LIN {X 0,Y 392.487,Z 448.569,A -85,B 0,C 180,E1 15700.156,E2 15700.156} C_VEL
LIN {X 0,Y 396.034,Z 422.526,A -85,B 0,C 180,E1 15700.091,E2 15700.091} C_VEL
LIN {X 0,Y 397.206,Z 415.686,A -85,B 0,C 180,E1 15700.071,E2 15700.071} C_VEL
LIN {X 0,Y 405.627,Z 392.982,A -85,B 0,C 180,E1 15699.396,E2 15699.396} C_VEL
LIN {X 0,Y 416.715,Z 367.074,A -85,B 0,C 180,E1 15698.867,E2 15698.867} C_VEL
LIN {X 0,Y 418.207,Z 363.431,A -85,B 0,C 180,E1 15698.784,E2 15698.784} C_VEL
LIN {X 0,Y 413.743,Z 355.491,A -85,B 0,C 180,E1 15697.429,E2 15697.429} C_VEL
LIN {X 0,Y 395.759,Z 367.716,A -85,B 0,C 180,E1 15695.526,E2 15695.526} C_VEL
LIN {X 0,Y 388.299,Z 373.214,A -85,B 0,C 180,E1 15694.685,E2 15694.685} C_VEL
LIN {X 0,Y 386.532,Z 374.791,A -85,B 0,C 180,E1 15694.506,E2 15694.506} C_VEL
LIN {X 0,Y 379.414,Z 383.98,A -85,B 0,C 180,E1 15694.055,E2 15694.055} C_VEL
LIN {X 0,Y 377.884,Z 385.781,A -85,B 0,C 180,E1 15693.937,E2 15693.937} C_VEL
LIN {X 0,Y 373.363,Z 392.757,A -85,B 0,C 180,E1 15693.757,E2 15693.757} C_VEL
LIN {X 0,Y 371.922,Z 395.3,A -85,B 0,C 180,E1 15693.628,E2 15693.628} C_VEL
LIN {X 0,Y 367.95,Z 408.603,A -85,B 0,C 180,E1 15693.013,E2 15693.013} C_VEL
LIN {X 0,Y 361.272,Z 436.616,A -85,B 0,C 180,E1 15692.192,E2 15692.192} C_VEL
LIN {X 0,Y 356.729,Z 450.848,A -85,B 0,C 180,E1 15691.567,E2 15691.567} C_VEL
LIN {X 0,Y 354.7,Z 456.048,A -85,B 0,C 180,E1 15691.213,E2 15691.213} C_VEL
LIN {X 0,Y 350.036,Z 511.042,A -85,B 0,C 180,E1 15689.32,E2 15689.32} C_VEL
LIN {X 0,Y 348.814,Z 540.503,A -85,B 0,C 180,E1 15688.156,E2 15688.156} C_VEL
LIN {X 0,Y 347.785,Z 558.819,A -85,B 0,C 180,E1 15687.108,E2 15687.108} C_VEL
LIN {X 0,Y 346.431,Z 575.545,A -85,B 0,C 180,E1 15685.836,E2 15685.836} C_VEL
LIN {X 0,Y 344.795,Z 591.161,A -85,B 0,C 180,E1 15684.316,E2 15684.316} C_VEL
LIN {X 0,Y 342.925,Z 605.58,A -85,B 0,C 180,E1 15682.545,E2 15682.545} C_VEL
LIN {X 0,Y 341.004,Z 618.295,A -85,B 0,C 180,E1 15680.6,E2 15680.6} C_VEL
LIN {X 0,Y 339.13,Z 628.932,A -85,B 0,C 180,E1 15678.567,E2 15678.567} C_VEL
LIN {X 0,Y 337.33,Z 638.29,A -85,B 0,C 180,E1 15676.354,E2 15676.354} C_VEL
LIN {X 0,Y 335.653,Z 646.221,A -85,B 0,C 180,E1 15673.962,E2 15673.962} C_VEL
LIN {X 0,Y 334.164,Z 652.657,A -85,B 0,C 180,E1 15671.389,E2 15671.389} C_VEL
LIN {X 0,Y 332.887,Z 657.506,A -85,B 0,C 180,E1 15668.637,E2 15668.637} C_VEL
LIN {X 0,Y 331.953,Z 660.524,A -85,B 0,C 180,E1 15665.877,E2 15665.877} C_VEL
LIN {X 0,Y 331.293,Z 661.723,A -85,B 0,C 180,E1 15663.114,E2 15663.114} C_VEL
LIN {X 0,Y 330.87,Z 661.148,A -85,B 0,C 180,E1 15660.173,E2 15660.173} C_VEL
LIN {X 0,Y 330.688,Z 658.902,A -85,B 0,C 180,E1 15657.4,E2 15657.4} C_VEL
LIN {X 0,Y 330.725,Z 654.896,A -85,B 0,C 180,E1 15654.622,E2 15654.622} C_VEL
LIN {X 0,Y 331.012,Z 649.083,A -85,B 0,C 180,E1 15651.838,E2 15651.838} C_VEL
LIN {X 0,Y 331.551,Z 641.849,A -85,B 0,C 180,E1 15649.223,E2 15649.223} C_VEL
LIN {X 0,Y 332.288,Z 633.259,A -85,B 0,C 180,E1 15646.78,E2 15646.78} C_VEL
LIN {X 0,Y 333.301,Z 622.56,A -85,B 0,C 180,E1 15644.336,E2 15644.336} C_VEL
LIN {X 0,Y 334.517,Z 610.39,A -85,B 0,C 180,E1 15642.069,E2 15642.069} C_VEL
LIN {X 0,Y 335.851,Z 596.537,A -85,B 0,C 180,E1 15639.978,E2 15639.978} C_VEL
LIN {X 0,Y 337.259,Z 580.898,A -85,B 0,C 180,E1 15638.065,E2 15638.065} C_VEL
LIN {X 0,Y 338.196,Z 569.28,A -85,B 0,C 180,E1 15636.891,E2 15636.891} C_VEL
LIN {X 0,Y 339.206,Z 569.951,A -85,B 0,C 180,E1 15636.55,E2 15636.55} C_VEL
LIN {X 0,Y 341.148,Z 569.562,A -85,B 0,C 180,E1 15636.142,E2 15636.142} C_VEL
LIN {X 0,Y 344.557,Z 567.21,A -85,B 0,C 180,E1 15635.671,E2 15635.671} C_VEL
LIN {X 0,Y 345.598,Z 566.259,A -85,B 0,C 180,E1 15635.561,E2 15635.561} C_VEL
LIN {X 0,Y 349.13,Z 565.085,A -85,B 0,C 180,E1 15634.921,E2 15634.921} C_VEL
LIN {X 0,Y 353.11,Z 562.349,A -85,B 0,C 180,E1 15634.416,E2 15634.416} C_VEL
LIN {X 0,Y 355.079,Z 560.666,A -85,B 0,C 180,E1 15634.211,E2 15634.211} C_VEL
LIN {X 0,Y 359.526,Z 558.324,A -85,B 0,C 180,E1 15633.578,E2 15633.578} C_VEL
LIN {X 0,Y 364.457,Z 554.315,A -85,B 0,C 180,E1 15633.077,E2 15633.077} C_VEL
LIN {X 0,Y 366.509,Z 552.398,A -85,B 0,C 180,E1 15632.897,E2 15632.897} C_VEL
LIN {X 0,Y 371.92,Z 548.521,A -85,B 0,C 180,E1 15632.283,E2 15632.283} C_VEL
LIN {X 0,Y 374.478,Z 546.267,A -85,B 0,C 180,E1 15632.046,E2 15632.046} C_VEL
LIN {X 0,Y 370.607,Z 566.083,A -85,B 0,C 180,E1 15630.625,E2 15630.625} C_VEL
LIN {X 0,Y 366.1,Z 585.225,A -85,B 0,C 180,E1 15628.923,E2 15628.923} C_VEL
LIN {X 0,Y 361.315,Z 603.126,A -85,B 0,C 180,E1 15626.981,E2 15626.981} C_VEL
LIN {X 0,Y 356.284,Z 620.142,A -85,B 0,C 180,E1 15624.751,E2 15624.751} C_VEL
LIN {X 0,Y 351.291,Z 635.867,A -85,B 0,C 180,E1 15622.269,E2 15622.269} C_VEL
LIN {X 0,Y 346.268,Z 650.875,A -85,B 0,C 180,E1 15619.414,E2 15619.414} C_VEL
LIN {X 0,Y 341.918,Z 663.648,A -85,B 0,C 180,E1 15616.488,E2 15616.488} C_VEL
LIN {X 0,Y 337.835,Z 675.827,A -85,B 0,C 180,E1 15613.132,E2 15613.132} C_VEL
LIN {X 0,Y 334.436,Z 686.527,A -85,B 0,C 180,E1 15609.525,E2 15609.525} C_VEL
LIN {X 0,Y 331.909,Z 695.291,A -85,B 0,C 180,E1 15605.869,E2 15605.869} C_VEL
LIN {X 0,Y 330.179,Z 702.285,A -85,B 0,C 180,E1 15602.207,E2 15602.207} C_VEL
LIN {X 0,Y 329.103,Z 707.622,A -85,B 0,C 180,E1 15598.489,E2 15598.489} C_VEL
LIN {X 0,Y 328.55,Z 711.353,A -85,B 0,C 180,E1 15594.833,E2 15594.833} C_VEL
LIN {X 0,Y 328.309,Z 713.66,A -85,B 0,C 180,E1 15591.249,E2 15591.249} C_VEL
LIN {X 0,Y 328.236,Z 714.499,A -85,B 0,C 180,E1 15587.735,E2 15587.735} C_VEL
LIN {X 0,Y 328.262,Z 713.981,A -85,B 0,C 180,E1 15584.104,E2 15584.104} C_VEL
LIN {X 0,Y 328.384,Z 712.133,A -85,B 0,C 180,E1 15580.527,E2 15580.527} C_VEL
LIN {X 0,Y 328.393,Z 711.979,A -85,B 0,C 180,E1 15580.342,E2 15580.342} C_VEL
LIN {X 0,Y 327.504,Z 710.953,A -85,B 0,C 180,E1 15579.009,E2 15579.009} C_VEL
LIN {X 0,Y 321.728,Z 707.66,A -85,B 0,C 180,E1 15575.334,E2 15575.334} C_VEL
LIN {X 0,Y 321.323,Z 706.322,A -85,B 0,C 180,E1 15574.266,E2 15574.266} C_VEL
LIN {X 0,Y 322.528,Z 700.31,A -85,B 0,C 180,E1 15570.533,E2 15570.533} C_VEL
LIN {X 0,Y 324.543,Z 692.213,A -85,B 0,C 180,E1 15566.645,E2 15566.645} C_VEL
LIN {X 0,Y 327.135,Z 683.135,A -85,B 0,C 180,E1 15563.154,E2 15563.154} C_VEL
LIN {X 0,Y 330.488,Z 672.221,A -85,B 0,C 180,E1 15559.718,E2 15559.718} C_VEL
LIN {X 0,Y 334.648,Z 659.116,A -85,B 0,C 180,E1 15556.348,E2 15556.348} C_VEL
LIN {X 0,Y 339.079,Z 645.119,A -85,B 0,C 180,E1 15553.38,E2 15553.38} C_VEL
LIN {X 0,Y 343.55,Z 630.595,A -85,B 0,C 180,E1 15550.8,E2 15550.8} C_VEL
LIN {X 0,Y 348.365,Z 614.201,A -85,B 0,C 180,E1 15548.358,E2 15548.358} C_VEL
LIN {X 0,Y 352.927,Z 597.492,A -85,B 0,C 180,E1 15546.279,E2 15546.279} C_VEL
LIN {X 0,Y 357.391,Z 579.198,A -85,B 0,C 180,E1 15544.391,E2 15544.391} C_VEL
LIN {X 0,Y 361.488,Z 559.757,A -85,B 0,C 180,E1 15542.757,E2 15542.757} C_VEL
LIN {X 0,Y 364.922,Z 540.309,A -85,B 0,C 180,E1 15541.438,E2 15541.438} C_VEL
LIN {X 0,Y 367.878,Z 519.528,A -85,B 0,C 180,E1 15540.33,E2 15540.33} C_VEL
LIN {X 0,Y 370.025,Z 498.949,A -85,B 0,C 180,E1 15539.504,E2 15539.504} C_VEL
LIN {X 0,Y 373.205,Z 458.095,A -85,B 0,C 180,E1 15538.359,E2 15538.359} C_VEL
LIN {X 0,Y 381.534,Z 354.699,A -85,B 0,C 180,E1 15535.843,E2 15535.843} C_VEL
LIN {X 0,Y 385.855,Z 290.048,A -85,B 0,C 180,E1 15534.392,E2 15534.392} C_VEL
LIN {X 0,Y 373.209,Z 274.366,A -85,B 0,C 180,E1 15531.534,E2 15531.534} C_VEL
LIN {X 0,Y 362.14,Z 261.496,A -85,B 0,C 180,E1 15528.797,E2 15528.797} C_VEL
LIN {X 0,Y 351.673,Z 250.184,A -85,B 0,C 180,E1 15525.94,E2 15525.94} C_VEL
LIN {X 0,Y 350.591,Z 248.929,A -85,B 0,C 180,E1 15525.479,E2 15525.479} C_VEL
LIN {X 0,Y 348.435,Z 244.814,A -85,B 0,C 180,E1 15523.687,E2 15523.687} C_VEL
LIN {X 0,Y 345.9,Z 240.181,A -85,B 0,C 180,E1 15521.449,E2 15521.449} C_VEL
LIN {X 0,Y 343.592,Z 235.82,A -85,B 0,C 180,E1 15519.16,E2 15519.16} C_VEL
LIN {X 0,Y 340.833,Z 231.357,A -85,B 0,C 180,E1 15516.222,E2 15516.222} C_VEL
LIN {X 0,Y 340.177,Z 230.148,A -85,B 0,C 180,E1 15515.383,E2 15515.383} C_VEL
LIN {X 0,Y 337.729,Z 226.321,A -85,B 0,C 180,E1 15512.144,E2 15512.144} C_VEL
LIN {X 0,Y 337.178,Z 224.904,A -85,B 0,C 180,E1 15511.02,E2 15511.02} C_VEL
LIN {X 0,Y 334.065,Z 219.475,A -85,B 0,C 180,E1 15502.803,E2 15502.803} C_VEL
LIN {X 0,Y 333.683,Z 219.259,A -85,B 0,C 180,E1 15496.718,E2 15496.718} C_VEL
LIN {X 0,Y 334.153,Z 219.886,A -85,B 0,C 180,E1 15494.193,E2 15494.193} C_VEL
LIN {X 0,Y 337.514,Z 225.321,A -85,B 0,C 180,E1 15486.293,E2 15486.293} C_VEL
LIN {X 0,Y 339.579,Z 229.521,A -85,B 0,C 180,E1 15483.039,E2 15483.039} C_VEL
LIN {X 0,Y 340.714,Z 230.864,A -85,B 0,C 180,E1 15481.85,E2 15481.85} C_VEL
LIN {X 0,Y 342.824,Z 234.937,A -85,B 0,C 180,E1 15479.332,E2 15479.332} C_VEL
LIN {X 0,Y 343.813,Z 236.632,A -85,B 0,C 180,E1 15478.334,E2 15478.334} C_VEL
LIN {X 0,Y 346.489,Z 241.285,A -85,B 0,C 180,E1 15475.864,E2 15475.864} C_VEL
LIN {X 0,Y 349.453,Z 246.993,A -85,B 0,C 180,E1 15473.264,E2 15473.264} C_VEL
LIN {X 0,Y 352.167,Z 252.01,A -85,B 0,C 180,E1 15471.181,E2 15471.181} C_VEL
LIN {X 0,Y 355.969,Z 259.17,A -85,B 0,C 180,E1 15468.497,E2 15468.497} C_VEL
LIN {X 0,Y 361.905,Z 271.338,A -85,B 0,C 180,E1 15464.62,E2 15464.62} C_VEL
LIN {X 0,Y 367.914,Z 284.797,A -85,B 0,C 180,E1 15460.967,E2 15460.967} C_VEL
LIN {X 0,Y 374.021,Z 299.419,A -85,B 0,C 180,E1 15457.526,E2 15457.526} C_VEL
LIN {X 0,Y 377.825,Z 309.539,A -85,B 0,C 180,E1 15455.405,E2 15455.405} C_VEL
LIN {X 0,Y 371.739,Z 345.671,A -85,B 0,C 180,E1 15451.746,E2 15451.746} C_VEL
LIN {X 0,Y 370.156,Z 368.005,A -85,B 0,C 180,E1 15449.201,E2 15449.201} C_VEL
LIN {X 0,Y 370.795,Z 387.836,A -85,B 0,C 180,E1 15446.712,E2 15446.712} C_VEL
LIN {X 0,Y 373.748,Z 407.381,A -85,B 0,C 180,E1 15444.041,E2 15444.041} C_VEL
LIN {X 0,Y 378.959,Z 425.383,A -85,B 0,C 180,E1 15441.392,E2 15441.392} C_VEL
LIN {X 0,Y 380.443,Z 428.811,A -85,B 0,C 180,E1 15440.943,E2 15440.943} C_VEL
LIN {X 0,Y 385.693,Z 438.336,A -85,B 0,C 180,E1 15439.863,E2 15439.863} C_VEL
LIN {X 0,Y 380.299,Z 469.554,A -85,B 0,C 180,E1 15439.844,E2 15439.844} C_VEL
LIN {X 0,Y 376.787,Z 493.447,A -85,B 0,C 180,E1 15439.502,E2 15439.502} C_VEL
LIN {X 0,Y 373.459,Z 519.124,A -85,B 0,C 180,E1 15438.728,E2 15438.728} C_VEL
LIN {X 0,Y 368.825,Z 547.178,A -85,B 0,C 180,E1 15437.623,E2 15437.623} C_VEL
LIN {X 0,Y 364.001,Z 572.411,A -85,B 0,C 180,E1 15436.331,E2 15436.331} C_VEL
LIN {X 0,Y 358.942,Z 596.768,A -85,B 0,C 180,E1 15434.74,E2 15434.74} C_VEL
LIN {X 0,Y 353.662,Z 620.524,A -85,B 0,C 180,E1 15432.831,E2 15432.831} C_VEL
LIN {X 0,Y 348.8,Z 641.281,A -85,B 0,C 180,E1 15430.812,E2 15430.812} C_VEL
LIN {X 0,Y 343.855,Z 660.827,A -85,B 0,C 180,E1 15428.482,E2 15428.482} C_VEL
LIN {X 0,Y 339.268,Z 678.112,A -85,B 0,C 180,E1 15426.011,E2 15426.011} C_VEL
LIN {X 0,Y 334.603,Z 695.333,A -85,B 0,C 180,E1 15423.048,E2 15423.048} C_VEL
LIN {X 0,Y 330.777,Z 709.483,A -85,B 0,C 180,E1 15420.117,E2 15420.117} C_VEL
LIN {X 0,Y 327.199,Z 723.351,A -85,B 0,C 180,E1 15416.692,E2 15416.692} C_VEL
LIN {X 0,Y 324.461,Z 734.858,A -85,B 0,C 180,E1 15413.231,E2 15413.231} C_VEL
LIN {X 0,Y 322.411,Z 744.868,A -85,B 0,C 180,E1 15409.568,E2 15409.568} C_VEL
LIN {X 0,Y 321.071,Z 753.191,A -85,B 0,C 180,E1 15405.719,E2 15405.719} C_VEL
LIN {X 0,Y 320.41,Z 759.339,A -85,B 0,C 180,E1 15402.068,E2 15402.068} C_VEL
LIN {X 0,Y 320.185,Z 763.743,A -85,B 0,C 180,E1 15398.439,E2 15398.439} C_VEL
LIN {X 0,Y 320.199,Z 766.573,A -85,B 0,C 180,E1 15394.836,E2 15394.836} C_VEL
LIN {X 0,Y 320.243,Z 767.835,A -85,B 0,C 180,E1 15391.431,E2 15391.431} C_VEL
LIN {X 0,Y 320.242,Z 767.696,A -85,B 0,C 180,E1 15388.032,E2 15388.032} C_VEL
LIN {X 0,Y 320.19,Z 766.069,A -85,B 0,C 180,E1 15384.445,E2 15384.445} C_VEL
LIN {X 0,Y 320.206,Z 762.931,A -85,B 0,C 180,E1 15380.836,E2 15380.836} C_VEL
LIN {X 0,Y 320.499,Z 758.218,A -85,B 0,C 180,E1 15377.203,E2 15377.203} C_VEL
LIN {X 0,Y 321.316,Z 751.453,A -85,B 0,C 180,E1 15373.364,E2 15373.364} C_VEL
LIN {X 0,Y 322.853,Z 742.799,A -85,B 0,C 180,E1 15369.515,E2 15369.515} C_VEL
LIN {X 0,Y 325.262,Z 731.977,A -85,B 0,C 180,E1 15365.674,E2 15365.674} C_VEL
LIN {X 0,Y 328.303,Z 720.191,A -85,B 0,C 180,E1 15362.227,E2 15362.227} C_VEL
LIN {X 0,Y 332.228,Z 706.136,A -85,B 0,C 180,E1 15358.825,E2 15358.825} C_VEL
LIN {X 0,Y 336.602,Z 691.156,A -85,B 0,C 180,E1 15355.793,E2 15355.793} C_VEL
LIN {X 0,Y 341.706,Z 673.731,A -85,B 0,C 180,E1 15352.867,E2 15352.867} C_VEL
LIN {X 0,Y 346.738,Z 656.164,A -85,B 0,C 180,E1 15350.41,E2 15350.41} C_VEL
LIN {X 0,Y 351.861,Z 637.171,A -85,B 0,C 180,E1 15348.213,E2 15348.213} C_VEL
LIN {X 0,Y 356.891,Z 617.213,A -85,B 0,C 180,E1 15346.312,E2 15346.312} C_VEL
LIN {X 0,Y 362.566,Z 593.122,A -85,B 0,C 180,E1 15344.417,E2 15344.417} C_VEL
LIN {X 0,Y 367.944,Z 568.826,A -85,B 0,C 180,E1 15342.883,E2 15342.883} C_VEL
LIN {X 0,Y 373.14,Z 543.519,A -85,B 0,C 180,E1 15341.616,E2 15341.616} C_VEL
LIN {X 0,Y 378.336,Z 514.4,A -85,B 0,C 180,E1 15340.487,E2 15340.487} C_VEL
LIN {X 0,Y 381.981,Z 490.052,A -85,B 0,C 180,E1 15339.765,E2 15339.765} C_VEL
LIN {X 0,Y 385.473,Z 466.122,A -85,B 0,C 180,E1 15339.371,E2 15339.371} C_VEL
LIN {X 0,Y 389.514,Z 434.671,A -85,B 0,C 180,E1 15339.144,E2 15339.144} C_VEL
LIN {X 0,Y 392.766,Z 412.557,A -85,B 0,C 180,E1 15339.122,E2 15339.122} C_VEL
LIN {X 0,Y 401.669,Z 389.192,A -85,B 0,C 180,E1 15338.464,E2 15338.464} C_VEL
LIN {X 0,Y 411.384,Z 366.3,A -85,B 0,C 180,E1 15337.993,E2 15337.993} C_VEL
LIN {X 0,Y 410.276,Z 364.543,A -85,B 0,C 180,E1 15337.668,E2 15337.668} C_VEL
LIN {X 0,Y 390.27,Z 378.406,A -85,B 0,C 180,E1 15335.56,E2 15335.56} C_VEL
LIN {X 0,Y 388.489,Z 379.968,A -85,B 0,C 180,E1 15335.386,E2 15335.386} C_VEL
LIN {X 0,Y 381.886,Z 388.423,A -85,B 0,C 180,E1 15334.986,E2 15334.986} C_VEL
LIN {X 0,Y 379.907,Z 391.219,A -85,B 0,C 180,E1 15334.89,E2 15334.89} C_VEL
LIN {X 0,Y 375.28,Z 398.265,A -85,B 0,C 180,E1 15334.645,E2 15334.645} C_VEL
LIN {X 0,Y 371.299,Z 411.381,A -85,B 0,C 180,E1 15334.063,E2 15334.063} C_VEL
LIN {X 0,Y 364.548,Z 439.135,A -85,B 0,C 180,E1 15333.274,E2 15333.274} C_VEL
LIN {X 0,Y 359.777,Z 453.854,A -85,B 0,C 180,E1 15332.65,E2 15332.65} C_VEL
LIN {X 0,Y 357.387,Z 459.804,A -85,B 0,C 180,E1 15332.312,E2 15332.312} C_VEL
LIN {X 0,Y 352.276,Z 475.72,A -85,B 0,C 180,E1 15331.864,E2 15331.864} C_VEL
LIN {X 0,Y 348.359,Z 485.195,A -85,B 0,C 180,E1 15331.407,E2 15331.407} C_VEL
LIN {X 0,Y 346.115,Z 489.605,A -85,B 0,C 180,E1 15331.04,E2 15331.04} C_VEL
LIN {X 0,Y 343.332,Z 527.625,A -85,B 0,C 180,E1 15329.608,E2 15329.608} C_VEL
LIN {X 0,Y 342.389,Z 548.043,A -85,B 0,C 180,E1 15328.662,E2 15328.662} C_VEL
LIN {X 0,Y 340.99,Z 567.202,A -85,B 0,C 180,E1 15327.41,E2 15327.41} C_VEL
LIN {X 0,Y 339.336,Z 583.333,A -85,B 0,C 180,E1 15326.013,E2 15326.013} C_VEL
LIN {X 0,Y 337.519,Z 598.174,A -85,B 0,C 180,E1 15324.409,E2 15324.409} C_VEL
LIN {X 0,Y 335.333,Z 612.593,A -85,B 0,C 180,E1 15322.432,E2 15322.432} C_VEL
LIN {X 0,Y 333.387,Z 623.729,A -85,B 0,C 180,E1 15320.541,E2 15320.541} C_VEL
LIN {X 0,Y 331.442,Z 633.701,A -85,B 0,C 180,E1 15318.466,E2 15318.466} C_VEL
LIN {X 0,Y 329.409,Z 642.917,A -85,B 0,C 180,E1 15316.034,E2 15316.034} C_VEL
LIN {X 0,Y 327.699,Z 650.162,A -85,B 0,C 180,E1 15313.587,E2 15313.587} C_VEL
LIN {X 0,Y 326.183,Z 655.968,A -85,B 0,C 180,E1 15310.955,E2 15310.955} C_VEL
LIN {X 0,Y 324.891,Z 660.181,A -85,B 0,C 180,E1 15308.138,E2 15308.138} C_VEL
LIN {X 0,Y 323.95,Z 662.571,A -85,B 0,C 180,E1 15305.312,E2 15305.312} C_VEL
LIN {X 0,Y 323.319,Z 663.266,A -85,B 0,C 180,E1 15302.481,E2 15302.481} C_VEL
LIN {X 0,Y 322.933,Z 662.196,A -85,B 0,C 180,E1 15299.645,E2 15299.645} C_VEL
LIN {X 0,Y 322.768,Z 659.22,A -85,B 0,C 180,E1 15296.625,E2 15296.625} C_VEL
LIN {X 0,Y 322.879,Z 654.596,A -85,B 0,C 180,E1 15293.746,E2 15293.746} C_VEL
LIN {X 0,Y 323.25,Z 648.157,A -85,B 0,C 180,E1 15290.923,E2 15290.923} C_VEL
LIN {X 0,Y 323.939,Z 639.593,A -85,B 0,C 180,E1 15288.064,E2 15288.064} C_VEL
LIN {X 0,Y 324.82,Z 630.078,A -85,B 0,C 180,E1 15285.561,E2 15285.561} C_VEL
LIN {X 0,Y 326.003,Z 618.281,A -85,B 0,C 180,E1 15283.06,E2 15283.06} C_VEL
LIN {X 0,Y 327.326,Z 605.363,A -85,B 0,C 180,E1 15280.829,E2 15280.829} C_VEL
LIN {X 0,Y 328.745,Z 590.679,A -85,B 0,C 180,E1 15278.78,E2 15278.78} C_VEL
LIN {X 0,Y 329.79,Z 579.388,A -85,B 0,C 180,E1 15277.447,E2 15277.447} C_VEL
LIN {X 0,Y 330.904,Z 579.966,A -85,B 0,C 180,E1 15277.058,E2 15277.058} C_VEL
LIN {X 0,Y 333.581,Z 579.142,A -85,B 0,C 180,E1 15276.506,E2 15276.506} C_VEL
LIN {X 0,Y 336.645,Z 577.059,A -85,B 0,C 180,E1 15276.082,E2 15276.082} C_VEL
LIN {X 0,Y 339.654,Z 576.354,A -85,B 0,C 180,E1 15275.476,E2 15275.476} C_VEL
LIN {X 0,Y 343.839,Z 573.887,A -85,B 0,C 180,E1 15274.877,E2 15274.877} C_VEL
LIN {X 0,Y 345.549,Z 572.843,A -85,B 0,C 180,E1 15274.643,E2 15274.643} C_VEL
LIN {X 0,Y 350.333,Z 570.614,A -85,B 0,C 180,E1 15273.926,E2 15273.926} C_VEL
LIN {X 0,Y 355.113,Z 567.108,A -85,B 0,C 180,E1 15273.404,E2 15273.404} C_VEL
LIN {X 0,Y 360.234,Z 564.331,A -85,B 0,C 180,E1 15272.743,E2 15272.743} C_VEL
LIN {X 0,Y 365.659,Z 560.04,A -85,B 0,C 180,E1 15272.21,E2 15272.21} C_VEL
LIN {X 0,Y 366.71,Z 559.079,A -85,B 0,C 180,E1 15272.122,E2 15272.122} C_VEL
LIN {X 0,Y 362.306,Z 578.303,A -85,B 0,C 180,E1 15270.54,E2 15270.54} C_VEL
LIN {X 0,Y 357.318,Z 597.116,A -85,B 0,C 180,E1 15268.635,E2 15268.635} C_VEL
LIN {X 0,Y 352.062,Z 614.673,A -85,B 0,C 180,E1 15266.465,E2 15266.465} C_VEL
LIN {X 0,Y 346.877,Z 630.625,A -85,B 0,C 180,E1 15264.094,E2 15264.094} C_VEL
LIN {X 0,Y 341.664,Z 645.762,A -85,B 0,C 180,E1 15261.386,E2 15261.386} C_VEL
LIN {X 0,Y 336.536,Z 660.118,A -85,B 0,C 180,E1 15258.278,E2 15258.278} C_VEL
LIN {X 0,Y 331.859,Z 673.17,A -85,B 0,C 180,E1 15254.832,E2 15254.832} C_VEL
LIN {X 0,Y 327.963,Z 684.385,A -85,B 0,C 180,E1 15251.188,E2 15251.188} C_VEL
LIN {X 0,Y 325.026,Z 693.514,A -85,B 0,C 180,E1 15247.525,E2 15247.525} C_VEL
LIN {X 0,Y 322.851,Z 701.167,A -85,B 0,C 180,E1 15243.667,E2 15243.667} C_VEL
LIN {X 0,Y 321.427,Z 707.263,A -85,B 0,C 180,E1 15239.644,E2 15239.644} C_VEL
LIN {X 0,Y 320.714,Z 711.396,A -85,B 0,C 180,E1 15235.879,E2 15235.879} C_VEL
LIN {X 0,Y 320.391,Z 713.935,A -85,B 0,C 180,E1 15232.186,E2 15232.186} C_VEL
LIN {X 0,Y 320.267,Z 715.102,A -85,B 0,C 180,E1 15228.362,E2 15228.362} C_VEL
LIN {X 0,Y 320.275,Z 714.911,A -85,B 0,C 180,E1 15224.833,E2 15224.833} C_VEL
LIN {X 0,Y 320.381,Z 713.228,A -85,B 0,C 180,E1 15221.157,E2 15221.157} C_VEL
LIN {X 0,Y 320.729,Z 710.026,A -85,B 0,C 180,E1 15217.344,E2 15217.344} C_VEL
LIN {X 0,Y 321.323,Z 706.322,A -85,B 0,C 180,E1 15214.266,E2 15214.266} C_VEL
LIN {X 0,Y 320.683,Z 704.566,A -85,B 0,C 180,E1 15212.921,E2 15212.921} C_VEL
LIN {X 0,Y 315.789,Z 699.114,A -85,B 0,C 180,E1 15209.219,E2 15209.219} C_VEL
LIN {X 0,Y 315.698,Z 697.08,A -85,B 0,C 180,E1 15208.168,E2 15208.168} C_VEL
LIN {X 0,Y 318.14,Z 688.482,A -85,B 0,C 180,E1 15204.409,E2 15204.409} C_VEL
LIN {X 0,Y 321.278,Z 678.498,A -85,B 0,C 180,E1 15200.868,E2 15200.868} C_VEL
LIN {X 0,Y 325.218,Z 666.505,A -85,B 0,C 180,E1 15197.392,E2 15197.392} C_VEL
LIN {X 0,Y 329.757,Z 652.902,A -85,B 0,C 180,E1 15194.164,E2 15194.164} C_VEL
LIN {X 0,Y 334.431,Z 638.592,A -85,B 0,C 180,E1 15191.343,E2 15191.343} C_VEL
LIN {X 0,Y 339.359,Z 622.825,A -85,B 0,C 180,E1 15188.753,E2 15188.753} C_VEL
LIN {X 0,Y 344.415,Z 605.469,A -85,B 0,C 180,E1 15186.383,E2 15186.383} C_VEL
LIN {X 0,Y 348.953,Z 588.504,A -85,B 0,C 180,E1 15184.455,E2 15184.455} C_VEL
LIN {X 0,Y 353.338,Z 570.024,A -85,B 0,C 180,E1 15182.715,E2 15182.715} C_VEL
LIN {X 0,Y 357.244,Z 550.406,A -85,B 0,C 180,E1 15181.224,E2 15181.224} C_VEL
LIN {X 0,Y 360.428,Z 530.954,A -85,B 0,C 180,E1 15180.044,E2 15180.044} C_VEL
LIN {X 0,Y 363.083,Z 509.821,A -85,B 0,C 180,E1 15179.051,E2 15179.051} C_VEL
LIN {X 0,Y 364.987,Z 487.926,A -85,B 0,C 180,E1 15178.301,E2 15178.301} C_VEL
LIN {X 0,Y 374.009,Z 382.48,A -85,B 0,C 180,E1 15175.587,E2 15175.587} C_VEL
LIN {X 0,Y 380.186,Z 300.146,A -85,B 0,C 180,E1 15173.711,E2 15173.711} C_VEL
LIN {X 0,Y 380.443,Z 294.212,A -85,B 0,C 180,E1 15173.562,E2 15173.562} C_VEL
LIN {X 0,Y 367.114,Z 277.751,A -85,B 0,C 180,E1 15170.424,E2 15170.424} C_VEL
LIN {X 0,Y 356.185,Z 265.217,A -85,B 0,C 180,E1 15167.586,E2 15167.586} C_VEL
LIN {X 0,Y 347.637,Z 256.092,A -85,B 0,C 180,E1 15165.152,E2 15165.152} C_VEL
LIN {X 0,Y 344.891,Z 253.099,A -85,B 0,C 180,E1 15164.269,E2 15164.269} C_VEL
LIN {X 0,Y 341.447,Z 246.68,A -85,B 0,C 180,E1 15161.186,E2 15161.186} C_VEL
LIN {X 0,Y 338.773,Z 241.89,A -85,B 0,C 180,E1 15158.518,E2 15158.518} C_VEL
LIN {X 0,Y 336.496,Z 237.638,A -85,B 0,C 180,E1 15155.788,E2 15155.788} C_VEL
LIN {X 0,Y 333.585,Z 232.935,A -85,B 0,C 180,E1 15151.839,E2 15151.839} C_VEL
LIN {X 0,Y 333.104,Z 231.762,A -85,B 0,C 180,E1 15150.855,E2 15150.855} C_VEL
LIN {X 0,Y 330.17,Z 226.462,A -85,B 0,C 180,E1 15142.807,E2 15142.807} C_VEL
LIN {X 0,Y 329.798,Z 226.253,A -85,B 0,C 180,E1 15136.66,E2 15136.66} C_VEL
LIN {X 0,Y 330.231,Z 226.896,A -85,B 0,C 180,E1 15134.197,E2 15134.197} C_VEL
LIN {X 0,Y 333.459,Z 232.29,A -85,B 0,C 180,E1 15126.37,E2 15126.37} C_VEL
LIN {X 0,Y 335.539,Z 236.432,A -85,B 0,C 180,E1 15123.075,E2 15123.075} C_VEL
LIN {X 0,Y 336.502,Z 237.597,A -85,B 0,C 180,E1 15122.044,E2 15122.044} C_VEL
LIN {X 0,Y 338.773,Z 241.872,A -85,B 0,C 180,E1 15119.324,E2 15119.324} C_VEL
LIN {X 0,Y 342.149,Z 248.093,A -85,B 0,C 180,E1 15115.979,E2 15115.979} C_VEL
LIN {X 0,Y 344.907,Z 253.41,A -85,B 0,C 180,E1 15113.509,E2 15113.509} C_VEL
LIN {X 0,Y 348.933,Z 260.791,A -85,B 0,C 180,E1 15110.434,E2 15110.434} C_VEL
LIN {X 0,Y 353.991,Z 271.358,A -85,B 0,C 180,E1 15106.775,E2 15106.775} C_VEL
LIN {X 0,Y 358.842,Z 281.681,A -85,B 0,C 180,E1 15103.656,E2 15103.656} C_VEL
LIN {X 0,Y 364.621,Z 295.138,A -85,B 0,C 180,E1 15100.122,E2 15100.122} C_VEL
LIN {X 0,Y 370.704,Z 310.369,A -85,B 0,C 180,E1 15096.642,E2 15096.642} C_VEL
LIN {X 0,Y 371.776,Z 313.221,A -85,B 0,C 180,E1 15096.04,E2 15096.04} C_VEL
LIN {X 0,Y 365.689,Z 347.948,A -85,B 0,C 180,E1 15092.479,E2 15092.479} C_VEL
LIN {X 0,Y 363.895,Z 369.961,A -85,B 0,C 180,E1 15089.941,E2 15089.941} C_VEL
LIN {X 0,Y 364.294,Z 390.2,A -85,B 0,C 180,E1 15087.372,E2 15087.372} C_VEL
LIN {X 0,Y 367.015,Z 410.03,A -85,B 0,C 180,E1 15084.626,E2 15084.626} C_VEL
LIN {X 0,Y 370.317,Z 422.699,A -85,B 0,C 180,E1 15082.81,E2 15082.81} C_VEL
LIN {X 0,Y 379.095,Z 440.038,A -85,B 0,C 180,E1 15080.851,E2 15080.851} C_VEL
LIN {X 0,Y 379.526,Z 441.187,A -85,B 0,C 180,E1 15080.75,E2 15080.75} C_VEL
LIN {X 0,Y 374.445,Z 471.137,A -85,B 0,C 180,E1 15080.702,E2 15080.702} C_VEL
LIN {X 0,Y 370.87,Z 494.696,A -85,B 0,C 180,E1 15080.327,E2 15080.327} C_VEL
LIN {X 0,Y 367.279,Z 521.054,A -85,B 0,C 180,E1 15079.498,E2 15079.498} C_VEL
LIN {X 0,Y 362.63,Z 548.051,A -85,B 0,C 180,E1 15078.409,E2 15078.409} C_VEL
LIN {X 0,Y 357.638,Z 573.082,A -85,B 0,C 180,E1 15077.095,E2 15077.095} C_VEL
LIN {X 0,Y 352.279,Z 598.081,A -85,B 0,C 180,E1 15075.431,E2 15075.431} C_VEL
LIN {X 0,Y 346.948,Z 621.241,A -85,B 0,C 180,E1 15073.532,E2 15073.532} C_VEL
LIN {X 0,Y 341.92,Z 641.7,A -85,B 0,C 180,E1 15071.49,E2 15071.49} C_VEL
LIN {X 0,Y 336.968,Z 660.665,A -85,B 0,C 180,E1 15069.199,E2 15069.199} C_VEL
LIN {X 0,Y 332.233,Z 677.665,A -85,B 0,C 180,E1 15066.719,E2 15066.719} C_VEL
LIN {X 0,Y 327.455,Z 694.606,A -85,B 0,C 180,E1 15063.76,E2 15063.76} C_VEL
LIN {X 0,Y 323.314,Z 709.191,A -85,B 0,C 180,E1 15060.681,E2 15060.681} C_VEL
LIN {X 0,Y 319.725,Z 722.384,A -85,B 0,C 180,E1 15057.361,E2 15057.361} C_VEL
LIN {X 0,Y 316.75,Z 734.191,A -85,B 0,C 180,E1 15053.736,E2 15053.736} C_VEL
LIN {X 0,Y 314.615,Z 744.017,A -85,B 0,C 180,E1 15050.073,E2 15050.073} C_VEL
LIN {X 0,Y 313.173,Z 752.41,A -85,B 0,C 180,E1 15046.126,E2 15046.126} C_VEL
LIN {X 0,Y 312.449,Z 758.59,A -85,B 0,C 180,E1 15042.38,E2 15042.38} C_VEL
LIN {X 0,Y 312.203,Z 763.024,A -85,B 0,C 180,E1 15038.657,E2 15038.657} C_VEL
LIN {X 0,Y 312.221,Z 765.885,A -85,B 0,C 180,E1 15034.96,E2 15034.96} C_VEL
LIN {X 0,Y 312.269,Z 767.165,A -85,B 0,C 180,E1 15031.468,E2 15031.468} C_VEL
LIN {X 0,Y 312.267,Z 767.048,A -85,B 0,C 180,E1 15027.981,E2 15027.981} C_VEL
LIN {X 0,Y 312.205,Z 765.43,A -85,B 0,C 180,E1 15024.302,E2 15024.302} C_VEL
LIN {X 0,Y 312.227,Z 762.197,A -85,B 0,C 180,E1 15020.51,E2 15020.51} C_VEL
LIN {X 0,Y 312.574,Z 757.314,A -85,B 0,C 180,E1 15016.684,E2 15016.684} C_VEL
LIN {X 0,Y 313.501,Z 750.476,A -85,B 0,C 180,E1 15012.746,E2 15012.746} C_VEL
LIN {X 0,Y 315.209,Z 741.746,A -85,B 0,C 180,E1 15008.8,E2 15008.8} C_VEL
LIN {X 0,Y 317.839,Z 730.839,A -85,B 0,C 180,E1 15004.869,E2 15004.869} C_VEL
LIN {X 0,Y 321.145,Z 718.986,A -85,B 0,C 180,E1 15001.349,E2 15001.349} C_VEL
LIN {X 0,Y 325.37,Z 704.835,A -85,B 0,C 180,E1 14997.884,E2 14997.884} C_VEL
LIN {X 0,Y 330.271,Z 689.076,A -85,B 0,C 180,E1 14994.673,E2 14994.673} C_VEL
LIN {X 0,Y 335.545,Z 672.017,A -85,B 0,C 180,E1 14991.807,E2 14991.807} C_VEL
LIN {X 0,Y 340.934,Z 654.122,A -85,B 0,C 180,E1 14989.304,E2 14989.304} C_VEL
LIN {X 0,Y 346.44,Z 634.68,A -85,B 0,C 180,E1 14987.068,E2 14987.068} C_VEL
LIN {X 0,Y 351.691,Z 614.331,A -85,B 0,C 180,E1 14985.165,E2 14985.165} C_VEL
LIN {X 0,Y 357.448,Z 590.834,A -85,B 0,C 180,E1 14983.341,E2 14983.341} C_VEL
LIN {X 0,Y 362.986,Z 566.648,A -85,B 0,C 180,E1 14981.831,E2 14981.831} C_VEL
LIN {X 0,Y 368.46,Z 540.638,A -85,B 0,C 180,E1 14980.552,E2 14980.552} C_VEL
LIN {X 0,Y 373.769,Z 511.333,A -85,B 0,C 180,E1 14979.433,E2 14979.433} C_VEL
LIN {X 0,Y 377.228,Z 489.257,A -85,B 0,C 180,E1 14978.791,E2 14978.791} C_VEL
LIN {X 0,Y 380.922,Z 465.007,A -85,B 0,C 180,E1 14978.393,E2 14978.393} C_VEL
LIN {X 0,Y 384.933,Z 434.534,A -85,B 0,C 180,E1 14978.172,E2 14978.172} C_VEL
LIN {X 0,Y 388.245,Z 411.211,A -85,B 0,C 180,E1 14978.16,E2 14978.16} C_VEL
LIN {X 0,Y 388.886,Z 408.239,A -85,B 0,C 180,E1 14978.116,E2 14978.116} C_VEL
LIN {X 0,Y 398.231,Z 384.459,A -85,B 0,C 180,E1 14977.495,E2 14977.495} C_VEL
LIN {X 0,Y 400.999,Z 377.684,A -85,B 0,C 180,E1 14977.339,E2 14977.339} C_VEL
LIN {X 0,Y 390.592,Z 385.061,A -85,B 0,C 180,E1 14976.258,E2 14976.258} C_VEL
LIN {X 0,Y 383.729,Z 393.859,A -85,B 0,C 180,E1 14975.869,E2 14975.869} C_VEL
LIN {X 0,Y 378.732,Z 401.472,A -85,B 0,C 180,E1 14975.634,E2 14975.634} C_VEL
LIN {X 0,Y 374.801,Z 414.175,A -85,B 0,C 180,E1 14975.091,E2 14975.091} C_VEL
LIN {X 0,Y 367.852,Z 442.149,A -85,B 0,C 180,E1 14974.316,E2 14974.316} C_VEL
LIN {X 0,Y 362.815,Z 457.305,A -85,B 0,C 180,E1 14973.688,E2 14973.688} C_VEL
LIN {X 0,Y 360.476,Z 463.091,A -85,B 0,C 180,E1 14973.39,E2 14973.39} C_VEL
LIN {X 0,Y 355.193,Z 479.029,A -85,B 0,C 180,E1 14972.95,E2 14972.95} C_VEL
LIN {X 0,Y 351.012,Z 488.872,A -85,B 0,C 180,E1 14972.487,E2 14972.487} C_VEL
LIN {X 0,Y 348.577,Z 493.632,A -85,B 0,C 180,E1 14972.169,E2 14972.169} C_VEL
LIN {X 0,Y 343.932,Z 505.264,A -85,B 0,C 180,E1 14971.821,E2 14971.821} C_VEL
LIN {X 0,Y 340.353,Z 512.12,A -85,B 0,C 180,E1 14971.404,E2 14971.404} C_VEL
LIN {X 0,Y 338.59,Z 514.862,A -85,B 0,C 180,E1 14971.102,E2 14971.102} C_VEL
LIN {X 0,Y 336.759,Z 544.959,A -85,B 0,C 180,E1 14969.785,E2 14969.785} C_VEL
LIN {X 0,Y 335.31,Z 564.08,A -85,B 0,C 180,E1 14968.593,E2 14968.593} C_VEL
LIN {X 0,Y 333.539,Z 580.864,A -85,B 0,C 180,E1 14967.203,E2 14967.203} C_VEL
LIN {X 0,Y 331.713,Z 595.13,A -85,B 0,C 180,E1 14965.724,E2 14965.724} C_VEL
LIN {X 0,Y 329.309,Z 610.465,A -85,B 0,C 180,E1 14963.722,E2 14963.722} C_VEL
LIN {X 0,Y 327.048,Z 622.691,A -85,B 0,C 180,E1 14961.71,E2 14961.71} C_VEL
LIN {X 0,Y 324.719,Z 633.887,A -85,B 0,C 180,E1 14959.423,E2 14959.423} C_VEL
LIN {X 0,Y 322.488,Z 643.45,A -85,B 0,C 180,E1 14956.944,E2 14956.944} C_VEL
LIN {X 0,Y 320.56,Z 650.865,A -85,B 0,C 180,E1 14954.449,E2 14954.449} C_VEL
LIN {X 0,Y 318.862,Z 656.901,A -85,B 0,C 180,E1 14951.76,E2 14951.76} C_VEL
LIN {X 0,Y 317.485,Z 661.133,A -85,B 0,C 180,E1 14949.059,E2 14949.059} C_VEL
LIN {X 0,Y 316.376,Z 663.813,A -85,B 0,C 180,E1 14946.168,E2 14946.168} C_VEL
LIN {X 0,Y 315.566,Z 664.751,A -85,B 0,C 180,E1 14943.087,E2 14943.087} C_VEL
LIN {X 0,Y 315.107,Z 663.891,A -85,B 0,C 180,E1 14940.181,E2 14940.181} C_VEL
LIN {X 0,Y 314.882,Z 661.298,A -85,B 0,C 180,E1 14937.269,E2 14937.269} C_VEL
LIN {X 0,Y 314.931,Z 656.647,A -85,B 0,C 180,E1 14934.168,E2 14934.168} C_VEL
LIN {X 0,Y 315.273,Z 650.373,A -85,B 0,C 180,E1 14931.243,E2 14931.243} C_VEL
LIN {X 0,Y 315.888,Z 642.563,A -85,B 0,C 180,E1 14928.497,E2 14928.497} C_VEL
LIN {X 0,Y 316.805,Z 632.68,A -85,B 0,C 180,E1 14925.748,E2 14925.748} C_VEL
LIN {X 0,Y 317.89,Z 622.057,A -85,B 0,C 180,E1 14923.367,E2 14923.367} C_VEL
LIN {X 0,Y 319.251,Z 609.021,A -85,B 0,C 180,E1 14920.99,E2 14920.99} C_VEL
LIN {X 0,Y 320.684,Z 594.932,A -85,B 0,C 180,E1 14918.892,E2 14918.892} C_VEL
LIN {X 0,Y 321.311,Z 588.664,A -85,B 0,C 180,E1 14918.073,E2 14918.073} C_VEL
LIN {X 0,Y 322.633,Z 589.225,A -85,B 0,C 180,E1 14917.592,E2 14917.592} C_VEL
LIN {X 0,Y 325.333,Z 588.369,A -85,B 0,C 180,E1 14917.025,E2 14917.025} C_VEL
LIN {X 0,Y 327.898,Z 586.927,A -85,B 0,C 180,E1 14916.613,E2 14916.613} C_VEL
LIN {X 0,Y 331.049,Z 586.177,A -85,B 0,C 180,E1 14915.937,E2 14915.937} C_VEL
LIN {X 0,Y 335.219,Z 583.897,A -85,B 0,C 180,E1 14915.317,E2 14915.317} C_VEL
LIN {X 0,Y 339.606,Z 582.357,A -85,B 0,C 180,E1 14914.541,E2 14914.541} C_VEL
LIN {X 0,Y 344.845,Z 579.366,A -85,B 0,C 180,E1 14913.85,E2 14913.85} C_VEL
LIN {X 0,Y 350.677,Z 576.512,A -85,B 0,C 180,E1 14913.041,E2 14913.041} C_VEL
LIN {X 0,Y 356.292,Z 572.807,A -85,B 0,C 180,E1 14912.416,E2 14912.416} C_VEL
LIN {X 0,Y 358.614,Z 571.729,A -85,B 0,C 180,E1 14912.109,E2 14912.109} C_VEL
LIN {X 0,Y 353.982,Z 589.397,A -85,B 0,C 180,E1 14910.457,E2 14910.457} C_VEL
LIN {X 0,Y 348.632,Z 607.409,A -85,B 0,C 180,E1 14908.407,E2 14908.407} C_VEL
LIN {X 0,Y 343.211,Z 623.965,A -85,B 0,C 180,E1 14906.128,E2 14906.128} C_VEL
LIN {X 0,Y 337.856,Z 639.176,A -85,B 0,C 180,E1 14903.607,E2 14903.607} C_VEL
LIN {X 0,Y 332.349,Z 654.019,A -85,B 0,C 180,E1 14900.641,E2 14900.641} C_VEL
LIN {X 0,Y 327.086,Z 667.866,A -85,B 0,C 180,E1 14897.263,E2 14897.263} C_VEL
LIN {X 0,Y 322.619,Z 679.705,A -85,B 0,C 180,E1 14893.719,E2 14893.719} C_VEL
LIN {X 0,Y 318.975,Z 689.847,A -85,B 0,C 180,E1 14889.986,E2 14889.986} C_VEL
LIN {X 0,Y 316.278,Z 698.026,A -85,B 0,C 180,E1 14886.24,E2 14886.24} C_VEL
LIN {X 0,Y 314.266,Z 705.118,A -85,B 0,C 180,E1 14882.095,E2 14882.095} C_VEL
LIN {X 0,Y 313.152,Z 710.085,A -85,B 0,C 180,E1 14878.2,E2 14878.2} C_VEL
LIN {X 0,Y 312.578,Z 713.527,A -85,B 0,C 180,E1 14874.265,E2 14874.265} C_VEL
LIN {X 0,Y 312.348,Z 715.299,A -85,B 0,C 180,E1 14870.618,E2 14870.618} C_VEL
LIN {X 0,Y 312.286,Z 715.836,A -85,B 0,C 180,E1 14866.797,E2 14866.797} C_VEL
LIN {X 0,Y 312.332,Z 714.968,A -85,B 0,C 180,E1 14863.138,E2 14863.138} C_VEL
LIN {X 0,Y 312.532,Z 712.69,A -85,B 0,C 180,E1 14859.391,E2 14859.391} C_VEL
LIN {X 0,Y 313.087,Z 708.869,A -85,B 0,C 180,E1 14855.498,E2 14855.498} C_VEL
LIN {X 0,Y 314.153,Z 703.474,A -85,B 0,C 180,E1 14851.642,E2 14851.642} C_VEL
LIN {X 0,Y 315.698,Z 697.08,A -85,B 0,C 180,E1 14848.168,E2 14848.168} C_VEL
LIN {X 0,Y 315.489,Z 694.504,A -85,B 0,C 180,E1 14846.839,E2 14846.839} C_VEL
LIN {X 0,Y 311.856,Z 687.289,A -85,B 0,C 180,E1 14843.244,E2 14843.244} C_VEL
LIN {X 0,Y 312.053,Z 684.44,A -85,B 0,C 180,E1 14842.137,E2 14842.137} C_VEL
LIN {X 0,Y 315.628,Z 673.923,A -85,B 0,C 180,E1 14838.673,E2 14838.673} C_VEL
LIN {X 0,Y 320.172,Z 660.855,A -85,B 0,C 180,E1 14835.163,E2 14835.163} C_VEL
LIN {X 0,Y 324.994,Z 646.881,A -85,B 0,C 180,E1 14832.082,E2 14832.082} C_VEL
LIN {X 0,Y 329.834,Z 632.366,A -85,B 0,C 180,E1 14829.412,E2 14829.412} C_VEL
LIN {X 0,Y 335.03,Z 615.969,A -85,B 0,C 180,E1 14826.893,E2 14826.893} C_VEL
LIN {X 0,Y 339.929,Z 599.241,A -85,B 0,C 180,E1 14824.755,E2 14824.755} C_VEL
LIN {X 0,Y 344.72,Z 580.961,A -85,B 0,C 180,E1 14822.818,E2 14822.818} C_VEL
LIN {X 0,Y 349.116,Z 561.57,A -85,B 0,C 180,E1 14821.146,E2 14821.146} C_VEL
LIN {X 0,Y 352.785,Z 542.074,A -85,B 0,C 180,E1 14819.797,E2 14819.797} C_VEL
LIN {X 0,Y 355.829,Z 521.988,A -85,B 0,C 180,E1 14818.702,E2 14818.702} C_VEL
LIN {X 0,Y 358.234,Z 500.303,A -85,B 0,C 180,E1 14817.815,E2 14817.815} C_VEL
LIN {X 0,Y 362.16,Z 455.324,A -85,B 0,C 180,E1 14816.514,E2 14816.514} C_VEL
LIN {X 0,Y 370.467,Z 361.308,A -85,B 0,C 180,E1 14814.156,E2 14814.156} C_VEL
LIN {X 0,Y 375.133,Z 298.571,A -85,B 0,C 180,E1 14812.726,E2 14812.726} C_VEL
LIN {X 0,Y 363.204,Z 283.732,A -85,B 0,C 180,E1 14809.812,E2 14809.812} C_VEL
LIN {X 0,Y 351.415,Z 269.995,A -85,B 0,C 180,E1 14806.633,E2 14806.633} C_VEL
LIN {X 0,Y 340.654,Z 258.641,A -85,B 0,C 180,E1 14803.38,E2 14803.38} C_VEL
LIN {X 0,Y 338.842,Z 256.816,A -85,B 0,C 180,E1 14802.714,E2 14802.714} C_VEL
LIN {X 0,Y 337.059,Z 253.253,A -85,B 0,C 180,E1 14800.964,E2 14800.964} C_VEL
LIN {X 0,Y 334.411,Z 248.464,A -85,B 0,C 180,E1 14798.238,E2 14798.238} C_VEL
LIN {X 0,Y 331.905,Z 243.78,A -85,B 0,C 180,E1 14795.127,E2 14795.127} C_VEL
LIN {X 0,Y 329.499,Z 239.755,A -85,B 0,C 180,E1 14791.667,E2 14791.667} C_VEL
LIN {X 0,Y 329.032,Z 238.62,A -85,B 0,C 180,E1 14790.686,E2 14790.686} C_VEL
LIN {X 0,Y 326.246,Z 233.433,A -85,B 0,C 180,E1 14782.708,E2 14782.708} C_VEL
LIN {X 0,Y 325.917,Z 233.25,A -85,B 0,C 180,E1 14776.578,E2 14776.578} C_VEL
LIN {X 0,Y 326.3,Z 233.796,A -85,B 0,C 180,E1 14774.372,E2 14774.372} C_VEL
LIN {X 0,Y 329.405,Z 239.252,A -85,B 0,C 180,E1 14766.449,E2 14766.449} C_VEL
LIN {X 0,Y 331.664,Z 243.518,A -85,B 0,C 180,E1 14762.938,E2 14762.938} C_VEL
LIN {X 0,Y 332.482,Z 244.945,A -85,B 0,C 180,E1 14761.896,E2 14761.896} C_VEL
LIN {X 0,Y 335.124,Z 249.788,A -85,B 0,C 180,E1 14758.804,E2 14758.804} C_VEL
LIN {X 0,Y 337.812,Z 254.885,A -85,B 0,C 180,E1 14756.097,E2 14756.097} C_VEL
LIN {X 0,Y 340.37,Z 259.828,A -85,B 0,C 180,E1 14753.761,E2 14753.761} C_VEL
LIN {X 0,Y 344.303,Z 267.24,A -85,B 0,C 180,E1 14750.641,E2 14750.641} C_VEL
LIN {X 0,Y 350.042,Z 279.23,A -85,B 0,C 180,E1 14746.455,E2 14746.455} C_VEL
LIN {X 0,Y 355.766,Z 292.19,A -85,B 0,C 180,E1 14742.669,E2 14742.669} C_VEL
LIN {X 0,Y 361.263,Z 305.745,A -85,B 0,C 180,E1 14739.252,E2 14739.252} C_VEL
LIN {X 0,Y 365.676,Z 317.38,A -85,B 0,C 180,E1 14736.643,E2 14736.643} C_VEL
LIN {X 0,Y 359.625,Z 350.665,A -85,B 0,C 180,E1 14733.185,E2 14733.185} C_VEL
LIN {X 0,Y 357.635,Z 373.381,A -85,B 0,C 180,E1 14730.525,E2 14730.525} C_VEL
LIN {X 0,Y 357.885,Z 393.393,A -85,B 0,C 180,E1 14727.94,E2 14727.94} C_VEL
LIN {X 0,Y 360.435,Z 413.251,A -85,B 0,C 180,E1 14725.149,E2 14725.149} C_VEL
LIN {X 0,Y 361.525,Z 417.746,A -85,B 0,C 180,E1 14724.543,E2 14724.543} C_VEL
LIN {X 0,Y 369.717,Z 436.157,A -85,B 0,C 180,E1 14722.52,E2 14722.52} C_VEL
LIN {X 0,Y 373.512,Z 443.874,A -85,B 0,C 180,E1 14721.655,E2 14721.655} C_VEL
LIN {X 0,Y 368.838,Z 471.534,A -85,B 0,C 180,E1 14721.591,E2 14721.591} C_VEL
LIN {X 0,Y 365.164,Z 495.051,A -85,B 0,C 180,E1 14721.199,E2 14721.199} C_VEL
LIN {X 0,Y 361.155,Z 523.128,A -85,B 0,C 180,E1 14720.291,E2 14720.291} C_VEL
LIN {X 0,Y 356.064,Z 550.802,A -85,B 0,C 180,E1 14719.12,E2 14719.12} C_VEL
LIN {X 0,Y 350.783,Z 576.355,A -85,B 0,C 180,E1 14717.726,E2 14717.726} C_VEL
LIN {X 0,Y 345.517,Z 599.948,A -85,B 0,C 180,E1 14716.1,E2 14716.1} C_VEL
LIN {X 0,Y 339.938,Z 623.152,A -85,B 0,C 180,E1 14714.138,E2 14714.138} C_VEL
LIN {X 0,Y 334.665,Z 643.87,A -85,B 0,C 180,E1 14712.008,E2 14712.008} C_VEL
LIN {X 0,Y 329.763,Z 661.658,A -85,B 0,C 180,E1 14709.774,E2 14709.774} C_VEL
LIN {X 0,Y 324.576,Z 679.575,A -85,B 0,C 180,E1 14707.075,E2 14707.075} C_VEL
LIN {X 0,Y 319.935,Z 695.22,A -85,B 0,C 180,E1 14704.231,E2 14704.231} C_VEL
LIN {X 0,Y 315.425,Z 710.482,A -85,B 0,C 180,E1 14700.898,E2 14700.898} C_VEL
LIN {X 0,Y 311.759,Z 723.289,A -85,B 0,C 180,E1 14697.505,E2 14697.505} C_VEL
LIN {X 0,Y 308.79,Z 734.687,A -85,B 0,C 180,E1 14693.875,E2 14693.875} C_VEL
LIN {X 0,Y 306.587,Z 744.343,A -85,B 0,C 180,E1 14690.077,E2 14690.077} C_VEL
LIN {X 0,Y 305.176,Z 752.321,A -85,B 0,C 180,E1 14686.17,E2 14686.17} C_VEL
LIN {X 0,Y 304.45,Z 758.335,A -85,B 0,C 180,E1 14682.325,E2 14682.325} C_VEL
LIN {X 0,Y 304.216,Z 762.85,A -85,B 0,C 180,E1 14678.315,E2 14678.315} C_VEL
LIN {X 0,Y 304.246,Z 765.418,A -85,B 0,C 180,E1 14674.712,E2 14674.712} C_VEL
LIN {X 0,Y 304.304,Z 766.547,A -85,B 0,C 180,E1 14671.129,E2 14671.129} C_VEL
LIN {X 0,Y 304.287,Z 766.291,A -85,B 0,C 180,E1 14667.551,E2 14667.551} C_VEL
LIN {X 0,Y 304.212,Z 764.546,A -85,B 0,C 180,E1 14663.773,E2 14663.773} C_VEL
LIN {X 0,Y 304.254,Z 761.276,A -85,B 0,C 180,E1 14659.969,E2 14659.969} C_VEL
LIN {X 0,Y 304.658,Z 756.413,A -85,B 0,C 180,E1 14656.138,E2 14656.138} C_VEL
LIN {X 0,Y 305.709,Z 749.517,A -85,B 0,C 180,E1 14652.095,E2 14652.095} C_VEL
LIN {X 0,Y 307.599,Z 740.707,A -85,B 0,C 180,E1 14648.049,E2 14648.049} C_VEL
LIN {X 0,Y 310.478,Z 729.739,A -85,B 0,C 180,E1 14644.025,E2 14644.025} C_VEL
LIN {X 0,Y 314.184,Z 717.384,A -85,B 0,C 180,E1 14640.318,E2 14640.318} C_VEL
LIN {X 0,Y 318.872,Z 702.78,A -85,B 0,C 180,E1 14636.719,E2 14636.719} C_VEL
LIN {X 0,Y 324.012,Z 687.248,A -85,B 0,C 180,E1 14633.556,E2 14633.556} C_VEL
LIN {X 0,Y 329.631,Z 670.048,A -85,B 0,C 180,E1 14630.657,E2 14630.657} C_VEL
LIN {X 0,Y 335.424,Z 651.68,A -85,B 0,C 180,E1 14628.108,E2 14628.108} C_VEL
LIN {X 0,Y 340.947,Z 632.964,A -85,B 0,C 180,E1 14625.97,E2 14625.97} C_VEL
LIN {X 0,Y 346.459,Z 612.507,A -85,B 0,C 180,E1 14624.061,E2 14624.061} C_VEL
LIN {X 0,Y 352.479,Z 588.639,A -85,B 0,C 180,E1 14622.237,E2 14622.237} C_VEL
LIN {X 0,Y 358.236,Z 564.17,A -85,B 0,C 180,E1 14620.731,E2 14620.731} C_VEL
LIN {X 0,Y 364.09,Z 537.152,A -85,B 0,C 180,E1 14619.433,E2 14619.433} C_VEL
LIN {X 0,Y 369.571,Z 507.146,A -85,B 0,C 180,E1 14618.309,E2 14618.309} C_VEL
LIN {X 0,Y 372.979,Z 486.353,A -85,B 0,C 180,E1 14617.745,E2 14617.745} C_VEL
LIN {X 0,Y 376.667,Z 462.976,A -85,B 0,C 180,E1 14617.381,E2 14617.381} C_VEL
LIN {X 0,Y 380.533,Z 434.194,A -85,B 0,C 180,E1 14617.173,E2 14617.173} C_VEL
LIN {X 0,Y 383.846,Z 410.779,A -85,B 0,C 180,E1 14617.17,E2 14617.17} C_VEL
LIN {X 0,Y 384.486,Z 405.745,A -85,B 0,C 180,E1 14617.15,E2 14617.15} C_VEL
LIN {X 0,Y 388.175,Z 396.103,A -85,B 0,C 180,E1 14616.881,E2 14616.881} C_VEL
LIN {X 0,Y 382.247,Z 404.825,A -85,B 0,C 180,E1 14616.599,E2 14616.599} C_VEL
LIN {X 0,Y 378.471,Z 416.833,A -85,B 0,C 180,E1 14616.101,E2 14616.101} C_VEL
LIN {X 0,Y 371.418,Z 444.72,A -85,B 0,C 180,E1 14615.352,E2 14615.352} C_VEL
LIN {X 0,Y 366.16,Z 460.291,A -85,B 0,C 180,E1 14614.732,E2 14614.732} C_VEL
LIN {X 0,Y 363.739,Z 466.329,A -85,B 0,C 180,E1 14614.446,E2 14614.446} C_VEL
LIN {X 0,Y 358.317,Z 482.25,A -85,B 0,C 180,E1 14614.017,E2 14614.017} C_VEL
LIN {X 0,Y 353.773,Z 492.531,A -85,B 0,C 180,E1 14613.554,E2 14613.554} C_VEL
LIN {X 0,Y 351.458,Z 497.132,A -85,B 0,C 180,E1 14613.278,E2 14613.278} C_VEL
LIN {X 0,Y 346.483,Z 509.079,A -85,B 0,C 180,E1 14612.917,E2 14612.917} C_VEL
LIN {X 0,Y 342.479,Z 516.509,A -85,B 0,C 180,E1 14612.469,E2 14612.469} C_VEL
LIN {X 0,Y 340.804,Z 519.222,A -85,B 0,C 180,E1 14612.252,E2 14612.252} C_VEL
LIN {X 0,Y 336.466,Z 528.316,A -85,B 0,C 180,E1 14611.934,E2 14611.934} C_VEL
LIN {X 0,Y 333.006,Z 533.717,A -85,B 0,C 180,E1 14611.495,E2 14611.495} C_VEL
LIN {X 0,Y 331.855,Z 535.405,A -85,B 0,C 180,E1 14611.276,E2 14611.276} C_VEL
LIN {X 0,Y 330.511,Z 554.544,A -85,B 0,C 180,E1 14610.257,E2 14610.257} C_VEL
LIN {X 0,Y 328.691,Z 572.946,A -85,B 0,C 180,E1 14608.925,E2 14608.925} C_VEL
LIN {X 0,Y 326.401,Z 590.534,A -85,B 0,C 180,E1 14607.255,E2 14607.255} C_VEL
LIN {X 0,Y 323.955,Z 605.778,A -85,B 0,C 180,E1 14605.404,E2 14605.404} C_VEL
LIN {X 0,Y 321.541,Z 618.668,A -85,B 0,C 180,E1 14603.454,E2 14603.454} C_VEL
LIN {X 0,Y 319.091,Z 630.084,A -85,B 0,C 180,E1 14601.314,E2 14601.314} C_VEL
LIN {X 0,Y 316.519,Z 640.797,A -85,B 0,C 180,E1 14598.796,E2 14598.796} C_VEL
LIN {X 0,Y 314.247,Z 649.12,A -85,B 0,C 180,E1 14596.259,E2 14596.259} C_VEL
LIN {X 0,Y 312.211,Z 656.013,A -85,B 0,C 180,E1 14593.519,E2 14593.519} C_VEL
LIN {X 0,Y 310.446,Z 661.286,A -85,B 0,C 180,E1 14590.578,E2 14590.578} C_VEL
LIN {X 0,Y 309.071,Z 664.59,A -85,B 0,C 180,E1 14587.621,E2 14587.621} C_VEL
LIN {X 0,Y 308.036,Z 666.178,A -85,B 0,C 180,E1 14584.467,E2 14584.467} C_VEL
LIN {X 0,Y 307.404,Z 665.903,A -85,B 0,C 180,E1 14581.49,E2 14581.49} C_VEL
LIN {X 0,Y 307.046,Z 663.874,A -85,B 0,C 180,E1 14578.507,E2 14578.507} C_VEL
LIN {X 0,Y 306.969,Z 659.911,A -85,B 0,C 180,E1 14575.352,E2 14575.352} C_VEL
LIN {X 0,Y 307.168,Z 654.647,A -85,B 0,C 180,E1 14572.518,E2 14572.518} C_VEL
LIN {X 0,Y 307.693,Z 647.104,A -85,B 0,C 180,E1 14569.515,E2 14569.515} C_VEL
LIN {X 0,Y 308.509,Z 638.023,A -85,B 0,C 180,E1 14566.696,E2 14566.696} C_VEL
LIN {X 0,Y 309.589,Z 627.385,A -85,B 0,C 180,E1 14564.066,E2 14564.066} C_VEL
LIN {X 0,Y 310.937,Z 614.86,A -85,B 0,C 180,E1 14561.553,E2 14561.553} C_VEL
LIN {X 0,Y 312.35,Z 601.596,A -85,B 0,C 180,E1 14559.382,E2 14559.382} C_VEL
LIN {X 0,Y 312.787,Z 597.396,A -85,B 0,C 180,E1 14558.775,E2 14558.775} C_VEL
LIN {X 0,Y 314.444,Z 597.882,A -85,B 0,C 180,E1 14558.158,E2 14558.158} C_VEL
LIN {X 0,Y 317.174,Z 596.895,A -85,B 0,C 180,E1 14557.576,E2 14557.576} C_VEL
LIN {X 0,Y 318.774,Z 596.053,A -85,B 0,C 180,E1 14557.306,E2 14557.306} C_VEL
LIN {X 0,Y 321.839,Z 595.543,A -85,B 0,C 180,E1 14556.567,E2 14556.567} C_VEL
LIN {X 0,Y 325.757,Z 593.696,A -85,B 0,C 180,E1 14555.906,E2 14555.906} C_VEL
LIN {X 0,Y 329.957,Z 592.443,A -85,B 0,C 180,E1 14555.088,E2 14555.088} C_VEL
LIN {X 0,Y 334.822,Z 590.165,A -85,B 0,C 180,E1 14554.341,E2 14554.341} C_VEL
LIN {X 0,Y 340.402,Z 587.767,A -85,B 0,C 180,E1 14553.482,E2 14553.482} C_VEL
LIN {X 0,Y 344.8,Z 585.393,A -85,B 0,C 180,E1 14552.917,E2 14552.917} C_VEL
LIN {X 0,Y 350.549,Z 582.618,A -85,B 0,C 180,E1 14552.154,E2 14552.154} C_VEL
LIN {X 0,Y 345.364,Z 600.349,A -85,B 0,C 180,E1 14550.289,E2 14550.289} C_VEL
LIN {X 0,Y 339.519,Z 618.095,A -85,B 0,C 180,E1 14548.011,E2 14548.011} C_VEL
LIN {X 0,Y 333.685,Z 634.271,A -85,B 0,C 180,E1 14545.489,E2 14545.489} C_VEL
LIN {X 0,Y 328.031,Z 649.042,A -85,B 0,C 180,E1 14542.707,E2 14542.707} C_VEL
LIN {X 0,Y 322.664,Z 662.553,A -85,B 0,C 180,E1 14539.635,E2 14539.635} C_VEL
LIN {X 0,Y 317.584,Z 675.189,A -85,B 0,C 180,E1 14536.135,E2 14536.135} C_VEL
LIN {X 0,Y 313.209,Z 686.283,A -85,B 0,C 180,E1 14532.344,E2 14532.344} C_VEL
LIN {X 0,Y 309.876,Z 695.296,A -85,B 0,C 180,E1 14528.517,E2 14528.517} C_VEL
LIN {X 0,Y 307.378,Z 702.853,A -85,B 0,C 180,E1 14524.472,E2 14524.472} C_VEL
LIN {X 0,Y 305.71,Z 708.847,A -85,B 0,C 180,E1 14520.244,E2 14520.244} C_VEL
LIN {X 0,Y 304.861,Z 712.89,A -85,B 0,C 180,E1 14516.281,E2 14516.281} C_VEL
LIN {X 0,Y 304.476,Z 715.37,A -85,B 0,C 180,E1 14512.392,E2 14512.392} C_VEL
LIN {X 0,Y 304.325,Z 716.426,A -85,B 0,C 180,E1 14508.584,E2 14508.584} C_VEL
LIN {X 0,Y 304.328,Z 716.226,A -85,B 0,C 180,E1 14504.849,E2 14504.849} C_VEL
LIN {X 0,Y 304.449,Z 714.536,A -85,B 0,C 180,E1 14500.981,E2 14500.981} C_VEL
LIN {X 0,Y 304.858,Z 711.317,A -85,B 0,C 180,E1 14496.97,E2 14496.97} C_VEL
LIN {X 0,Y 305.739,Z 706.602,A -85,B 0,C 180,E1 14493,E2 14493} C_VEL
LIN {X 0,Y 307.278,Z 700.283,A -85,B 0,C 180,E1 14489.068,E2 14489.068} C_VEL
LIN {X 0,Y 309.584,Z 692.179,A -85,B 0,C 180,E1 14485.183,E2 14485.183} C_VEL
LIN {X 0,Y 312.053,Z 684.44,A -85,B 0,C 180,E1 14482.137,E2 14482.137} C_VEL
LIN {X 0,Y 312.255,Z 681.101,A -85,B 0,C 180,E1 14480.858,E2 14480.858} C_VEL
LIN {X 0,Y 309.918,Z 672.416,A -85,B 0,C 180,E1 14477.532,E2 14477.532} C_VEL
LIN {X 0,Y 310.506,Z 668.469,A -85,B 0,C 180,E1 14476.299,E2 14476.299} C_VEL
LIN {X 0,Y 315.273,Z 655.362,A -85,B 0,C 180,E1 14473.036,E2 14473.036} C_VEL
LIN {X 0,Y 320.31,Z 641.202,A -85,B 0,C 180,E1 14470.108,E2 14470.108} C_VEL
LIN {X 0,Y 325.602,Z 625.604,A -85,B 0,C 180,E1 14467.428,E2 14467.428} C_VEL
LIN {X 0,Y 330.833,Z 609.072,A -85,B 0,C 180,E1 14465.064,E2 14465.064} C_VEL
LIN {X 0,Y 335.866,Z 591.693,A -85,B 0,C 180,E1 14463.001,E2 14463.001} C_VEL
LIN {X 0,Y 340.748,Z 572.583,A -85,B 0,C 180,E1 14461.139,E2 14461.139} C_VEL
LIN {X 0,Y 344.925,Z 553.154,A -85,B 0,C 180,E1 14459.613,E2 14459.613} C_VEL
LIN {X 0,Y 348.323,Z 533.907,A -85,B 0,C 180,E1 14458.408,E2 14458.408} C_VEL
LIN {X 0,Y 351.179,Z 513.005,A -85,B 0,C 180,E1 14457.391,E2 14457.391} C_VEL
LIN {X 0,Y 353.314,Z 490.612,A -85,B 0,C 180,E1 14456.591,E2 14456.591} C_VEL
LIN {X 0,Y 362.176,Z 396.746,A -85,B 0,C 180,E1 14454.062,E2 14454.062} C_VEL
LIN {X 0,Y 368.852,Z 317.379,A -85,B 0,C 180,E1 14452.186,E2 14452.186} C_VEL
LIN {X 0,Y 369.763,Z 302.732,A -85,B 0,C 180,E1 14451.833,E2 14451.833} C_VEL
LIN {X 0,Y 356.895,Z 286.651,A -85,B 0,C 180,E1 14448.541,E2 14448.541} C_VEL
LIN {X 0,Y 346.193,Z 274.55,A -85,B 0,C 180,E1 14445.511,E2 14445.511} C_VEL
LIN {X 0,Y 337.994,Z 265.737,A -85,B 0,C 180,E1 14442.933,E2 14442.933} C_VEL
LIN {X 0,Y 333.27,Z 260.838,A -85,B 0,C 180,E1 14441.303,E2 14441.303} C_VEL
LIN {X 0,Y 330.177,Z 255.179,A -85,B 0,C 180,E1 14438.062,E2 14438.062} C_VEL
LIN {X 0,Y 327.586,Z 250.411,A -85,B 0,C 180,E1 14434.804,E2 14434.804} C_VEL
LIN {X 0,Y 325.358,Z 246.322,A -85,B 0,C 180,E1 14431.315,E2 14431.315} C_VEL
LIN {X 0,Y 324.823,Z 245.37,A -85,B 0,C 180,E1 14430.32,E2 14430.32} C_VEL
LIN {X 0,Y 322.33,Z 240.408,A -85,B 0,C 180,E1 14422.622,E2 14422.622} C_VEL
LIN {X 0,Y 322.047,Z 240.258,A -85,B 0,C 180,E1 14416.412,E2 14416.412} C_VEL
LIN {X 0,Y 322.378,Z 240.811,A -85,B 0,C 180,E1 14414.367,E2 14414.367} C_VEL
LIN {X 0,Y 325.296,Z 245.955,A -85,B 0,C 180,E1 14406.708,E2 14406.708} C_VEL
LIN {X 0,Y 327.461,Z 250.252,A -85,B 0,C 180,E1 14403.151,E2 14403.151} C_VEL
LIN {X 0,Y 328.277,Z 251.667,A -85,B 0,C 180,E1 14402.095,E2 14402.095} C_VEL
LIN {X 0,Y 330.849,Z 256.533,A -85,B 0,C 180,E1 14398.962,E2 14398.962} C_VEL
LIN {X 0,Y 333.329,Z 261.287,A -85,B 0,C 180,E1 14396.389,E2 14396.389} C_VEL
LIN {X 0,Y 335.838,Z 266.246,A -85,B 0,C 180,E1 14394.019,E2 14394.019} C_VEL
LIN {X 0,Y 339.472,Z 273.253,A -85,B 0,C 180,E1 14391.02,E2 14391.02} C_VEL
LIN {X 0,Y 344.15,Z 283.357,A -85,B 0,C 180,E1 14387.415,E2 14387.415} C_VEL
LIN {X 0,Y 348.799,Z 293.723,A -85,B 0,C 180,E1 14384.198,E2 14384.198} C_VEL
LIN {X 0,Y 354.121,Z 306.673,A -85,B 0,C 180,E1 14380.711,E2 14380.711} C_VEL
LIN {X 0,Y 359.666,Z 321.146,A -85,B 0,C 180,E1 14377.312,E2 14377.312} C_VEL
LIN {X 0,Y 353.632,Z 353.266,A -85,B 0,C 180,E1 14373.927,E2 14373.927} C_VEL
LIN {X 0,Y 351.429,Z 376.231,A -85,B 0,C 180,E1 14371.199,E2 14371.199} C_VEL
LIN {X 0,Y 351.546,Z 397.178,A -85,B 0,C 180,E1 14368.445,E2 14368.445} C_VEL
LIN {X 0,Y 353.344,Z 412.596,A -85,B 0,C 180,E1 14366.296,E2 14366.296} C_VEL
LIN {X 0,Y 360.419,Z 430.93,A -85,B 0,C 180,E1 14364.344,E2 14364.344} C_VEL
LIN {X 0,Y 367.63,Z 446.525,A -85,B 0,C 180,E1 14362.581,E2 14362.581} C_VEL
LIN {X 0,Y 363.332,Z 471.642,A -85,B 0,C 180,E1 14362.505,E2 14362.505} C_VEL
LIN {X 0,Y 359.566,Z 495.025,A -85,B 0,C 180,E1 14362.103,E2 14362.103} C_VEL
LIN {X 0,Y 355.542,Z 522.063,A -85,B 0,C 180,E1 14361.215,E2 14361.215} C_VEL
LIN {X 0,Y 350.2,Z 550.433,A -85,B 0,C 180,E1 14360.01,E2 14360.01} C_VEL
LIN {X 0,Y 344.761,Z 575.988,A -85,B 0,C 180,E1 14358.607,E2 14358.607} C_VEL
LIN {X 0,Y 339.04,Z 600.645,A -85,B 0,C 180,E1 14356.878,E2 14356.878} C_VEL
LIN {X 0,Y 333.182,Z 624.224,A -85,B 0,C 180,E1 14354.847,E2 14354.847} C_VEL
LIN {X 0,Y 328.057,Z 643.632,A -85,B 0,C 180,E1 14352.817,E2 14352.817} C_VEL
LIN {X 0,Y 322.596,Z 662.688,A -85,B 0,C 180,E1 14350.374,E2 14350.374} C_VEL
LIN {X 0,Y 317.503,Z 679.497,A -85,B 0,C 180,E1 14347.775,E2 14347.775} C_VEL
LIN {X 0,Y 312.293,Z 696.263,A -85,B 0,C 180,E1 14344.632,E2 14344.632} C_VEL
LIN {X 0,Y 308.004,Z 710.138,A -85,B 0,C 180,E1 14341.51,E2 14341.51} C_VEL
LIN {X 0,Y 303.973,Z 723.591,A -85,B 0,C 180,E1 14337.845,E2 14337.845} C_VEL
LIN {X 0,Y 300.899,Z 734.807,A -85,B 0,C 180,E1 14334.124,E2 14334.124} C_VEL
LIN {X 0,Y 298.512,Z 744.912,A -85,B 0,C 180,E1 14329.977,E2 14329.977} C_VEL
LIN {X 0,Y 297.127,Z 752.523,A -85,B 0,C 180,E1 14326.018,E2 14326.018} C_VEL
LIN {X 0,Y 296.411,Z 758.584,A -85,B 0,C 180,E1 14321.874,E2 14321.874} C_VEL
LIN {X 0,Y 296.233,Z 762.646,A -85,B 0,C 180,E1 14317.954,E2 14317.954} C_VEL
LIN {X 0,Y 296.283,Z 765.061,A -85,B 0,C 180,E1 14314.064,E2 14314.064} C_VEL
LIN {X 0,Y 296.334,Z 765.927,A -85,B 0,C 180,E1 14310.386,E2 14310.386} C_VEL
LIN {X 0,Y 296.294,Z 765.416,A -85,B 0,C 180,E1 14306.711,E2 14306.711} C_VEL
LIN {X 0,Y 296.224,Z 763.456,A -85,B 0,C 180,E1 14302.905,E2 14302.905} C_VEL
LIN {X 0,Y 296.328,Z 759.812,A -85,B 0,C 180,E1 14298.911,E2 14298.911} C_VEL
LIN {X 0,Y 296.92,Z 754.33,A -85,B 0,C 180,E1 14294.772,E2 14294.772} C_VEL
LIN {X 0,Y 298.264,Z 747.041,A -85,B 0,C 180,E1 14290.617,E2 14290.617} C_VEL
LIN {X 0,Y 300.552,Z 737.736,A -85,B 0,C 180,E1 14286.471,E2 14286.471} C_VEL
LIN {X 0,Y 303.742,Z 726.899,A -85,B 0,C 180,E1 14282.557,E2 14282.557} C_VEL
LIN {X 0,Y 307.768,Z 714.542,A -85,B 0,C 180,E1 14278.898,E2 14278.898} C_VEL
LIN {X 0,Y 312.813,Z 699.897,A -85,B 0,C 180,E1 14275.322,E2 14275.322} C_VEL
LIN {X 0,Y 318.218,Z 684.485,A -85,B 0,C 180,E1 14272.214,E2 14272.214} C_VEL
LIN {X 0,Y 324.264,Z 666.921,A -85,B 0,C 180,E1 14269.295,E2 14269.295} C_VEL
LIN {X 0,Y 330.222,Z 648.858,A -85,B 0,C 180,E1 14266.82,E2 14266.82} C_VEL
LIN {X 0,Y 336.055,Z 629.714,A -85,B 0,C 180,E1 14264.676,E2 14264.676} C_VEL
LIN {X 0,Y 341.619,Z 609.696,A -85,B 0,C 180,E1 14262.847,E2 14262.847} C_VEL
LIN {X 0,Y 347.926,Z 585.429,A -85,B 0,C 180,E1 14261.03,E2 14261.03} C_VEL
LIN {X 0,Y 353.929,Z 560.459,A -85,B 0,C 180,E1 14259.535,E2 14259.535} C_VEL
LIN {X 0,Y 359.889,Z 533.461,A -85,B 0,C 180,E1 14258.282,E2 14258.282} C_VEL
LIN {X 0,Y 365.423,Z 503.516,A -85,B 0,C 180,E1 14257.18,E2 14257.18} C_VEL
LIN {X 0,Y 369.417,Z 480.242,A -85,B 0,C 180,E1 14256.605,E2 14256.605} C_VEL
LIN {X 0,Y 373.921,Z 451.479,A -85,B 0,C 180,E1 14256.241,E2 14256.241} C_VEL
LIN {X 0,Y 373.879,Z 451.428,A -85,B 0,C 180,E1 14256.229,E2 14256.229} C_VEL
LIN {X 0,Y 368.426,Z 466.174,A -85,B 0,C 180,E1 14255.611,E2 14255.611} C_VEL
LIN {X 0,Y 366.887,Z 470.337,A -85,B 0,C 180,E1 14255.466,E2 14255.466} C_VEL
LIN {X 0,Y 361.23,Z 486.303,A -85,B 0,C 180,E1 14255.036,E2 14255.036} C_VEL
LIN {X 0,Y 356.438,Z 496.758,A -85,B 0,C 180,E1 14254.564,E2 14254.564} C_VEL
LIN {X 0,Y 354.506,Z 500.628,A -85,B 0,C 180,E1 14254.361,E2 14254.361} C_VEL
LIN {X 0,Y 349.156,Z 512.898,A -85,B 0,C 180,E1 14253.995,E2 14253.995} C_VEL
LIN {X 0,Y 344.664,Z 520.913,A -85,B 0,C 180,E1 14253.522,E2 14253.522} C_VEL
LIN {X 0,Y 343.27,Z 523.326,A -85,B 0,C 180,E1 14253.376,E2 14253.376} C_VEL
LIN {X 0,Y 338.73,Z 532.428,A -85,B 0,C 180,E1 14253.037,E2 14253.037} C_VEL
LIN {X 0,Y 334.974,Z 538.133,A -85,B 0,C 180,E1 14252.599,E2 14252.599} C_VEL
LIN {X 0,Y 333.645,Z 540.127,A -85,B 0,C 180,E1 14252.44,E2 14252.44} C_VEL
LIN {X 0,Y 329.88,Z 546.863,A -85,B 0,C 180,E1 14252.136,E2 14252.136} C_VEL
LIN {X 0,Y 326.769,Z 551.074,A -85,B 0,C 180,E1 14251.719,E2 14251.719} C_VEL
LIN {X 0,Y 325.415,Z 552.671,A -85,B 0,C 180,E1 14251.463,E2 14251.463} C_VEL
LIN {X 0,Y 323.565,Z 570.061,A -85,B 0,C 180,E1 14250.244,E2 14250.244} C_VEL
LIN {X 0,Y 321.296,Z 586.739,A -85,B 0,C 180,E1 14248.737,E2 14248.737} C_VEL
LIN {X 0,Y 318.831,Z 601.523,A -85,B 0,C 180,E1 14247.046,E2 14247.046} C_VEL
LIN {X 0,Y 316.258,Z 614.891,A -85,B 0,C 180,E1 14245.164,E2 14245.164} C_VEL
LIN {X 0,Y 313.62,Z 626.816,A -85,B 0,C 180,E1 14243.087,E2 14243.087} C_VEL
LIN {X 0,Y 310.686,Z 638.539,A -85,B 0,C 180,E1 14240.526,E2 14240.526} C_VEL
LIN {X 0,Y 308.077,Z 647.649,A -85,B 0,C 180,E1 14237.957,E2 14237.957} C_VEL
LIN {X 0,Y 305.693,Z 655.284,A -85,B 0,C 180,E1 14235.168,E2 14235.168} C_VEL
LIN {X 0,Y 303.723,Z 660.951,A -85,B 0,C 180,E1 14232.355,E2 14232.355} C_VEL
LIN {X 0,Y 302.016,Z 664.997,A -85,B 0,C 180,E1 14229.335,E2 14229.335} C_VEL
LIN {X 0,Y 300.723,Z 667.297,A -85,B 0,C 180,E1 14226.208,E2 14226.208} C_VEL
LIN {X 0,Y 299.878,Z 667.783,A -85,B 0,C 180,E1 14223.249,E2 14223.249} C_VEL
LIN {X 0,Y 299.329,Z 666.547,A -85,B 0,C 180,E1 14220.191,E2 14220.191} C_VEL
LIN {X 0,Y 299.059,Z 663.377,A -85,B 0,C 180,E1 14216.933,E2 14216.933} C_VEL
LIN {X 0,Y 299.12,Z 658.599,A -85,B 0,C 180,E1 14213.859,E2 14213.859} C_VEL
LIN {X 0,Y 299.497,Z 651.864,A -85,B 0,C 180,E1 14210.778,E2 14210.778} C_VEL
LIN {X 0,Y 300.187,Z 643.644,A -85,B 0,C 180,E1 14207.886,E2 14207.886} C_VEL
LIN {X 0,Y 301.135,Z 634,A -85,B 0,C 180,E1 14205.186,E2 14205.186} C_VEL
LIN {X 0,Y 302.423,Z 622.03,A -85,B 0,C 180,E1 14202.49,E2 14202.49} C_VEL
LIN {X 0,Y 303.876,Z 608.941,A -85,B 0,C 180,E1 14200.089,E2 14200.089} C_VEL
LIN {X 0,Y 304.278,Z 605.504,A -85,B 0,C 180,E1 14199.514,E2 14199.514} C_VEL
LIN {X 0,Y 305.732,Z 605.994,A -85,B 0,C 180,E1 14198.915,E2 14198.915} C_VEL
LIN {X 0,Y 308.287,Z 605.241,A -85,B 0,C 180,E1 14198.3,E2 14198.3} C_VEL
LIN {X 0,Y 309.774,Z 604.553,A -85,B 0,C 180,E1 14198.011,E2 14198.011} C_VEL
LIN {X 0,Y 312.701,Z 604.174,A -85,B 0,C 180,E1 14197.238,E2 14197.238} C_VEL
LIN {X 0,Y 316.365,Z 602.705,A -85,B 0,C 180,E1 14196.532,E2 14196.532} C_VEL
LIN {X 0,Y 320.444,Z 601.673,A -85,B 0,C 180,E1 14195.66,E2 14195.66} C_VEL
LIN {X 0,Y 324.427,Z 600.024,A -85,B 0,C 180,E1 14194.971,E2 14194.971} C_VEL
LIN {X 0,Y 329.517,Z 598.211,A -85,B 0,C 180,E1 14194.09,E2 14194.09} C_VEL
LIN {X 0,Y 332.866,Z 596.634,A -85,B 0,C 180,E1 14193.604,E2 14193.604} C_VEL
LIN {X 0,Y 339.39,Z 593.938,A -85,B 0,C 180,E1 14192.639,E2 14192.639} C_VEL
LIN {X 0,Y 342.592,Z 592.264,A -85,B 0,C 180,E1 14192.247,E2 14192.247} C_VEL
LIN {X 0,Y 336.703,Z 610.344,A -85,B 0,C 180,E1 14190.125,E2 14190.125} C_VEL
LIN {X 0,Y 330.834,Z 626.663,A -85,B 0,C 180,E1 14187.804,E2 14187.804} C_VEL
LIN {X 0,Y 325.008,Z 641.669,A -85,B 0,C 180,E1 14185.226,E2 14185.226} C_VEL
LIN {X 0,Y 318.976,Z 656.318,A -85,B 0,C 180,E1 14182.178,E2 14182.178} C_VEL
LIN {X 0,Y 313.237,Z 669.849,A -85,B 0,C 180,E1 14178.732,E2 14178.732} C_VEL
LIN {X 0,Y 308.153,Z 681.794,A -85,B 0,C 180,E1 14174.98,E2 14174.98} C_VEL
LIN {X 0,Y 304.084,Z 691.718,A -85,B 0,C 180,E1 14171.119,E2 14171.119} C_VEL
LIN {X 0,Y 300.963,Z 699.927,A -85,B 0,C 180,E1 14167.123,E2 14167.123} C_VEL
LIN {X 0,Y 298.684,Z 706.781,A -85,B 0,C 180,E1 14162.834,E2 14162.834} C_VEL
LIN {X 0,Y 297.326,Z 711.842,A -85,B 0,C 180,E1 14158.524,E2 14158.524} C_VEL
LIN {X 0,Y 296.687,Z 715.08,A -85,B 0,C 180,E1 14154.489,E2 14154.489} C_VEL
LIN {X 0,Y 296.409,Z 716.757,A -85,B 0,C 180,E1 14150.538,E2 14150.538} C_VEL
LIN {X 0,Y 296.34,Z 717.099,A -85,B 0,C 180,E1 14146.465,E2 14146.465} C_VEL
LIN {X 0,Y 296.399,Z 716.148,A -85,B 0,C 180,E1 14142.666,E2 14142.666} C_VEL
LIN {X 0,Y 296.659,Z 713.684,A -85,B 0,C 180,E1 14138.724,E2 14138.724} C_VEL
LIN {X 0,Y 297.346,Z 709.665,A -85,B 0,C 180,E1 14134.629,E2 14134.629} C_VEL
LIN {X 0,Y 298.635,Z 704.109,A -85,B 0,C 180,E1 14130.576,E2 14130.576} C_VEL
LIN {X 0,Y 300.683,Z 696.873,A -85,B 0,C 180,E1 14126.569,E2 14126.569} C_VEL
LIN {X 0,Y 303.617,Z 687.8,A -85,B 0,C 180,E1 14122.621,E2 14122.621} C_VEL
LIN {X 0,Y 307.08,Z 677.877,A -85,B 0,C 180,E1 14119.115,E2 14119.115} C_VEL
LIN {X 0,Y 310.506,Z 668.469,A -85,B 0,C 180,E1 14116.299,E2 14116.299} C_VEL
LIN {X 0,Y 311.168,Z 664.355,A -85,B 0,C 180,E1 14115.091,E2 14115.091} C_VEL
LIN {X 0,Y 309.936,Z 653.273,A -85,B 0,C 180,E1 14111.763,E2 14111.763} C_VEL
LIN {X 0,Y 310.841,Z 649.169,A -85,B 0,C 180,E1 14110.799,E2 14110.799} C_VEL
LIN {X 0,Y 315.969,Z 635.003,A -85,B 0,C 180,E1 14108.075,E2 14108.075} C_VEL
LIN {X 0,Y 321.727,Z 618.201,A -85,B 0,C 180,E1 14105.39,E2 14105.39} C_VEL
LIN {X 0,Y 326.975,Z 601.553,A -85,B 0,C 180,E1 14103.19,E2 14103.19} C_VEL
LIN {X 0,Y 331.896,Z 584.188,A -85,B 0,C 180,E1 14101.282,E2 14101.282} C_VEL
LIN {X 0,Y 336.798,Z 564.14,A -85,B 0,C 180,E1 14099.493,E2 14099.493} C_VEL
LIN {X 0,Y 340.939,Z 543.661,A -85,B 0,C 180,E1 14098.039,E2 14098.039} C_VEL
LIN {X 0,Y 344.125,Z 523.819,A -85,B 0,C 180,E1 14096.941,E2 14096.941} C_VEL
LIN {X 0,Y 346.582,Z 503.14,A -85,B 0,C 180,E1 14096.073,E2 14096.073} C_VEL
LIN {X 0,Y 350.859,Z 458.864,A -85,B 0,C 180,E1 14094.73,E2 14094.73} C_VEL
LIN {X 0,Y 359.379,Z 371.163,A -85,B 0,C 180,E1 14092.455,E2 14092.455} C_VEL
LIN {X 0,Y 364.621,Z 307.147,A -85,B 0,C 180,E1 14090.963,E2 14090.963} C_VEL
LIN {X 0,Y 353.211,Z 292.854,A -85,B 0,C 180,E1 14087.935,E2 14087.935} C_VEL
LIN {X 0,Y 342.342,Z 280.309,A -85,B 0,C 180,E1 14084.74,E2 14084.74} C_VEL
LIN {X 0,Y 333.943,Z 271.465,A -85,B 0,C 180,E1 14082.005,E2 14082.005} C_VEL
LIN {X 0,Y 329.195,Z 266.699,A -85,B 0,C 180,E1 14080.312,E2 14080.312} C_VEL
LIN {X 0,Y 327.247,Z 264.66,A -85,B 0,C 180,E1 14079.459,E2 14079.459} C_VEL
LIN {X 0,Y 325.906,Z 261.848,A -85,B 0,C 180,E1 14077.85,E2 14077.85} C_VEL
LIN {X 0,Y 323.461,Z 257.225,A -85,B 0,C 180,E1 14074.665,E2 14074.665} C_VEL
LIN {X 0,Y 321.269,Z 253.104,A -85,B 0,C 180,E1 14071.107,E2 14071.107} C_VEL
LIN {X 0,Y 320.587,Z 252.087,A -85,B 0,C 180,E1 14069.884,E2 14069.884} C_VEL
LIN {X 0,Y 318.411,Z 247.381,A -85,B 0,C 180,E1 14062.526,E2 14062.526} C_VEL
LIN {X 0,Y 318.149,Z 247.244,A -85,B 0,C 180,E1 14056.431,E2 14056.431} C_VEL
LIN {X 0,Y 318.461,Z 247.829,A -85,B 0,C 180,E1 14054.362,E2 14054.362} C_VEL
LIN {X 0,Y 321.248,Z 252.914,A -85,B 0,C 180,E1 14046.793,E2 14046.793} C_VEL
LIN {X 0,Y 323.585,Z 257.334,A -85,B 0,C 180,E1 14043.012,E2 14043.012} C_VEL
LIN {X 0,Y 326.456,Z 262.938,A -85,B 0,C 180,E1 14039.299,E2 14039.299} C_VEL
LIN {X 0,Y 329.002,Z 268.07,A -85,B 0,C 180,E1 14036.516,E2 14036.516} C_VEL
LIN {X 0,Y 331.482,Z 273.055,A -85,B 0,C 180,E1 14034.114,E2 14034.114} C_VEL
LIN {X 0,Y 334.862,Z 279.684,A -85,B 0,C 180,E1 14031.241,E2 14031.241} C_VEL
LIN {X 0,Y 340.174,Z 291.239,A -85,B 0,C 180,E1 14027.093,E2 14027.093} C_VEL
LIN {X 0,Y 345.689,Z 304.266,A -85,B 0,C 180,E1 14023.188,E2 14023.188} C_VEL
LIN {X 0,Y 351.316,Z 318.798,A -85,B 0,C 180,E1 14019.446,E2 14019.446} C_VEL
LIN {X 0,Y 353.641,Z 325.28,A -85,B 0,C 180,E1 14017.956,E2 14017.956} C_VEL
LIN {X 0,Y 347.592,Z 356.481,A -85,B 0,C 180,E1 14014.622,E2 14014.622} C_VEL
LIN {X 0,Y 345.234,Z 379.564,A -85,B 0,C 180,E1 14011.831,E2 14011.831} C_VEL
LIN {X 0,Y 345.217,Z 400.627,A -85,B 0,C 180,E1 14009.016,E2 14009.016} C_VEL
LIN {X 0,Y 345.942,Z 408.114,A -85,B 0,C 180,E1 14007.995,E2 14007.995} C_VEL
LIN {X 0,Y 352.505,Z 427.486,A -85,B 0,C 180,E1 14005.98,E2 14005.98} C_VEL
LIN {X 0,Y 360.722,Z 446.514,A -85,B 0,C 180,E1 14003.815,E2 14003.815} C_VEL
LIN {X 0,Y 361.873,Z 449.093,A -85,B 0,C 180,E1 14003.527,E2 14003.527} C_VEL
LIN {X 0,Y 357.892,Z 471.934,A -85,B 0,C 180,E1 14003.445,E2 14003.445} C_VEL
LIN {X 0,Y 353.91,Z 495.938,A -85,B 0,C 180,E1 14003.011,E2 14003.011} C_VEL
LIN {X 0,Y 349.53,Z 523.789,A -85,B 0,C 180,E1 14002.06,E2 14002.06} C_VEL
LIN {X 0,Y 344.158,Z 551.327,A -85,B 0,C 180,E1 14000.868,E2 14000.868} C_VEL
LIN {X 0,Y 338.402,Z 577.164,A -85,B 0,C 180,E1 13999.406,E2 13999.406} C_VEL
LIN {X 0,Y 332.572,Z 601.576,A -85,B 0,C 180,E1 13997.667,E2 13997.667} C_VEL
LIN {X 0,Y 326.642,Z 624.816,A -85,B 0,C 180,E1 13995.642,E2 13995.642} C_VEL
LIN {X 0,Y 321.302,Z 644.067,A -85,B 0,C 180,E1 13993.573,E2 13993.573} C_VEL
LIN {X 0,Y 315.849,Z 662.424,A -85,B 0,C 180,E1 13991.182,E2 13991.182} C_VEL
LIN {X 0,Y 310.363,Z 679.716,A -85,B 0,C 180,E1 13988.445,E2 13988.445} C_VEL
LIN {X 0,Y 305.056,Z 696.156,A -85,B 0,C 180,E1 13985.302,E2 13985.302} C_VEL
LIN {X 0,Y 300.369,Z 710.514,A -85,B 0,C 180,E1 13981.956,E2 13981.956} C_VEL
LIN {X 0,Y 296.242,Z 723.732,A -85,B 0,C 180,E1 13978.248,E2 13978.248} C_VEL
LIN {X 0,Y 292.972,Z 735.079,A -85,B 0,C 180,E1 13974.327,E2 13974.327} C_VEL
LIN {X 0,Y 290.642,Z 744.486,A -85,B 0,C 180,E1 13970.332,E2 13970.332} C_VEL
LIN {X 0,Y 289.184,Z 752.028,A -85,B 0,C 180,E1 13966.263,E2 13966.263} C_VEL
LIN {X 0,Y 288.431,Z 758.073,A -85,B 0,C 180,E1 13962.004,E2 13962.004} C_VEL
LIN {X 0,Y 288.251,Z 762.077,A -85,B 0,C 180,E1 13957.975,E2 13957.975} C_VEL
LIN {X 0,Y 288.307,Z 764.374,A -85,B 0,C 180,E1 13954.176,E2 13954.176} C_VEL
LIN {X 0,Y 288.362,Z 765.263,A -85,B 0,C 180,E1 13950.397,E2 13950.397} C_VEL
LIN {X 0,Y 288.314,Z 764.77,A -85,B 0,C 180,E1 13946.62,E2 13946.62} C_VEL
LIN {X 0,Y 288.237,Z 762.876,A -85,B 0,C 180,E1 13942.789,E2 13942.789} C_VEL
LIN {X 0,Y 288.34,Z 759.435,A -85,B 0,C 180,E1 13938.802,E2 13938.802} C_VEL
LIN {X 0,Y 288.962,Z 754.039,A -85,B 0,C 180,E1 13934.547,E2 13934.547} C_VEL
LIN {X 0,Y 290.385,Z 746.852,A -85,B 0,C 180,E1 13930.279,E2 13930.279} C_VEL
LIN {X 0,Y 292.668,Z 738.192,A -85,B 0,C 180,E1 13926.226,E2 13926.226} C_VEL
LIN {X 0,Y 296.17,Z 726.988,A -85,B 0,C 180,E1 13922.013,E2 13922.013} C_VEL
LIN {X 0,Y 300.412,Z 714.828,A -85,B 0,C 180,E1 13918.273,E2 13918.273} C_VEL
LIN {X 0,Y 305.704,Z 700.352,A -85,B 0,C 180,E1 13914.626,E2 13914.626} C_VEL
LIN {X 0,Y 311.708,Z 684.202,A -85,B 0,C 180,E1 13911.281,E2 13911.281} C_VEL
LIN {X 0,Y 317.869,Z 667.32,A -85,B 0,C 180,E1 13908.417,E2 13908.417} C_VEL
LIN {X 0,Y 324.523,Z 648.076,A -85,B 0,C 180,E1 13905.745,E2 13905.745} C_VEL
LIN {X 0,Y 330.672,Z 628.883,A -85,B 0,C 180,E1 13903.583,E2 13903.583} C_VEL
LIN {X 0,Y 336.438,Z 608.88,A -85,B 0,C 180,E1 13901.759,E2 13901.759} C_VEL
LIN {X 0,Y 342.979,Z 584.501,A -85,B 0,C 180,E1 13899.941,E2 13899.941} C_VEL
LIN {X 0,Y 349.505,Z 558.155,A -85,B 0,C 180,E1 13898.384,E2 13898.384} C_VEL
LIN {X 0,Y 355.8,Z 530.261,A -85,B 0,C 180,E1 13897.118,E2 13897.118} C_VEL
LIN {X 0,Y 361.48,Z 499.886,A -85,B 0,C 180,E1 13896.029,E2 13896.029} C_VEL
LIN {X 0,Y 362.328,Z 494.801,A -85,B 0,C 180,E1 13895.868,E2 13895.868} C_VEL
LIN {X 0,Y 357.706,Z 504.035,A -85,B 0,C 180,E1 13895.426,E2 13895.426} C_VEL
LIN {X 0,Y 352.008,Z 516.715,A -85,B 0,C 180,E1 13895.05,E2 13895.05} C_VEL
LIN {X 0,Y 346.98,Z 525.298,A -85,B 0,C 180,E1 13894.563,E2 13894.563} C_VEL
LIN {X 0,Y 341.166,Z 536.339,A -85,B 0,C 180,E1 13894.14,E2 13894.14} C_VEL
LIN {X 0,Y 336.64,Z 543.065,A -85,B 0,C 180,E1 13893.636,E2 13893.636} C_VEL
LIN {X 0,Y 331.385,Z 551.881,A -85,B 0,C 180,E1 13893.203,E2 13893.203} C_VEL
LIN {X 0,Y 327.556,Z 556.714,A -85,B 0,C 180,E1 13892.703,E2 13892.703} C_VEL
LIN {X 0,Y 322.486,Z 564.131,A -85,B 0,C 180,E1 13892.174,E2 13892.174} C_VEL
LIN {X 0,Y 319.523,Z 567.365,A -85,B 0,C 180,E1 13891.715,E2 13891.715} C_VEL
LIN {X 0,Y 318.711,Z 568.329,A -85,B 0,C 180,E1 13891.542,E2 13891.542} C_VEL
LIN {X 0,Y 316.266,Z 584.992,A -85,B 0,C 180,E1 13890.071,E2 13890.071} C_VEL
LIN {X 0,Y 313.462,Z 600.736,A -85,B 0,C 180,E1 13888.313,E2 13888.313} C_VEL
LIN {X 0,Y 310.557,Z 614.575,A -85,B 0,C 180,E1 13886.378,E2 13886.378} C_VEL
LIN {X 0,Y 307.535,Z 627.268,A -85,B 0,C 180,E1 13884.182,E2 13884.182} C_VEL
LIN {X 0,Y 304.522,Z 638.338,A -85,B 0,C 180,E1 13881.778,E2 13881.778} C_VEL
LIN {X 0,Y 301.44,Z 648.497,A -85,B 0,C 180,E1 13878.969,E2 13878.969} C_VEL
LIN {X 0,Y 298.833,Z 656.044,A -85,B 0,C 180,E1 13876.204,E2 13876.204} C_VEL
LIN {X 0,Y 296.564,Z 662.056,A -85,B 0,C 180,E1 13873.253,E2 13873.253} C_VEL
LIN {X 0,Y 294.654,Z 666.3,A -85,B 0,C 180,E1 13870.163,E2 13870.163} C_VEL
LIN {X 0,Y 293.201,Z 668.673,A -85,B 0,C 180,E1 13867.051,E2 13867.051} C_VEL
LIN {X 0,Y 292.127,Z 669.318,A -85,B 0,C 180,E1 13863.728,E2 13863.728} C_VEL
LIN {X 0,Y 291.495,Z 668.135,A -85,B 0,C 180,E1 13860.589,E2 13860.589} C_VEL
LIN {X 0,Y 291.172,Z 665.217,A -85,B 0,C 180,E1 13857.441,E2 13857.441} C_VEL
LIN {X 0,Y 291.17,Z 660.565,A -85,B 0,C 180,E1 13854.284,E2 13854.284} C_VEL
LIN {X 0,Y 291.476,Z 654.495,A -85,B 0,C 180,E1 13851.318,E2 13851.318} C_VEL
LIN {X 0,Y 292.161,Z 646.014,A -85,B 0,C 180,E1 13848.177,E2 13848.177} C_VEL
LIN {X 0,Y 293.182,Z 635.753,A -85,B 0,C 180,E1 13845.18,E2 13845.18} C_VEL
LIN {X 0,Y 294.491,Z 623.827,A -85,B 0,C 180,E1 13842.411,E2 13842.411} C_VEL
LIN {X 0,Y 295.739,Z 613.26,A -85,B 0,C 180,E1 13840.342,E2 13840.342} C_VEL
LIN {X 0,Y 297.125,Z 613.691,A -85,B 0,C 180,E1 13839.719,E2 13839.719} C_VEL
LIN {X 0,Y 300.282,Z 612.677,A -85,B 0,C 180,E1 13838.923,E2 13838.923} C_VEL
LIN {X 0,Y 304.306,Z 612.04,A -85,B 0,C 180,E1 13837.798,E2 13837.798} C_VEL
LIN {X 0,Y 307.067,Z 611.095,A -85,B 0,C 180,E1 13837.201,E2 13837.201} C_VEL
LIN {X 0,Y 311.453,Z 610.027,A -85,B 0,C 180,E1 13836.198,E2 13836.198} C_VEL
LIN {X 0,Y 313.909,Z 609.116,A -85,B 0,C 180,E1 13835.739,E2 13835.739} C_VEL
LIN {X 0,Y 318.837,Z 607.692,A -85,B 0,C 180,E1 13834.754,E2 13834.754} C_VEL
LIN {X 0,Y 322.724,Z 606.224,A -85,B 0,C 180,E1 13834.097,E2 13834.097} C_VEL
LIN {X 0,Y 329.062,Z 603.844,A -85,B 0,C 180,E1 13833.08,E2 13833.08} C_VEL
LIN {X 0,Y 334.41,Z 601.75,A -85,B 0,C 180,E1 13832.292,E2 13832.292} C_VEL
LIN {X 0,Y 328.533,Z 618.314,A -85,B 0,C 180,E1 13830.155,E2 13830.155} C_VEL
LIN {X 0,Y 322.132,Z 634.675,A -85,B 0,C 180,E1 13827.593,E2 13827.593} C_VEL
LIN {X 0,Y 315.578,Z 650.231,A -85,B 0,C 180,E1 13824.618,E2 13824.618} C_VEL
LIN {X 0,Y 309.353,Z 664.314,A -85,B 0,C 180,E1 13821.312,E2 13821.312} C_VEL
LIN {X 0,Y 303.5,Z 677.289,A -85,B 0,C 180,E1 13817.558,E2 13817.558} C_VEL
LIN {X 0,Y 298.603,Z 688.247,A -85,B 0,C 180,E1 13813.613,E2 13813.613} C_VEL
LIN {X 0,Y 294.655,Z 697.594,A -85,B 0,C 180,E1 13809.387,E2 13809.387} C_VEL
LIN {X 0,Y 291.849,Z 704.93,A -85,B 0,C 180,E1 13805.139,E2 13805.139} C_VEL
LIN {X 0,Y 290.011,Z 710.529,A -85,B 0,C 180,E1 13800.854,E2 13800.854} C_VEL
LIN {X 0,Y 288.986,Z 714.556,A -85,B 0,C 180,E1 13796.509,E2 13796.509} C_VEL
LIN {X 0,Y 288.55,Z 716.926,A -85,B 0,C 180,E1 13792.406,E2 13792.406} C_VEL
LIN {X 0,Y 288.38,Z 717.792,A -85,B 0,C 180,E1 13788.392,E2 13788.392} C_VEL
LIN {X 0,Y 288.392,Z 717.329,A -85,B 0,C 180,E1 13784.251,E2 13784.251} C_VEL
LIN {X 0,Y 288.559,Z 715.511,A -85,B 0,C 180,E1 13780.179,E2 13780.179} C_VEL
LIN {X 0,Y 289.06,Z 712.208,A -85,B 0,C 180,E1 13776.156,E2 13776.156} C_VEL
LIN {X 0,Y 290.212,Z 707.007,A -85,B 0,C 180,E1 13771.777,E2 13771.777} C_VEL
LIN {X 0,Y 292.073,Z 700.4,A -85,B 0,C 180,E1 13767.646,E2 13767.646} C_VEL
LIN {X 0,Y 294.824,Z 692.057,A -85,B 0,C 180,E1 13763.575,E2 13763.575} C_VEL
LIN {X 0,Y 298.538,Z 681.794,A -85,B 0,C 180,E1 13759.581,E2 13759.581} C_VEL
LIN {X 0,Y 303.081,Z 669.716,A -85,B 0,C 180,E1 13755.794,E2 13755.794} C_VEL
LIN {X 0,Y 307.786,Z 657.305,A -85,B 0,C 180,E1 13752.611,E2 13752.611} C_VEL
LIN {X 0,Y 310.841,Z 649.169,A -85,B 0,C 180,E1 13750.799,E2 13750.799} C_VEL
LIN {X 0,Y 311.847,Z 644.377,A -85,B 0,C 180,E1 13749.689,E2 13749.689} C_VEL
LIN {X 0,Y 311.452,Z 632.184,A -85,B 0,C 180,E1 13746.746,E2 13746.746} C_VEL
LIN {X 0,Y 312.549,Z 626.774,A -85,B 0,C 180,E1 13745.743,E2 13745.743} C_VEL
LIN {X 0,Y 318.219,Z 610.028,A -85,B 0,C 180,E1 13743.301,E2 13743.301} C_VEL
LIN {X 0,Y 323.624,Z 592.462,A -85,B 0,C 180,E1 13741.186,E2 13741.186} C_VEL
LIN {X 0,Y 328.413,Z 574.954,A -85,B 0,C 180,E1 13739.441,E2 13739.441} C_VEL
LIN {X 0,Y 333.108,Z 554.685,A -85,B 0,C 180,E1 13737.806,E2 13737.806} C_VEL
LIN {X 0,Y 336.965,Z 534.053,A -85,B 0,C 180,E1 13736.502,E2 13736.502} C_VEL
LIN {X 0,Y 339.841,Z 513.692,A -85,B 0,C 180,E1 13735.516,E2 13735.516} C_VEL
LIN {X 0,Y 342.681,Z 485.631,A -85,B 0,C 180,E1 13734.531,E2 13734.531} C_VEL
LIN {X 0,Y 351.985,Z 396.054,A -85,B 0,C 180,E1 13732.069,E2 13732.069} C_VEL
LIN {X 0,Y 358.788,Z 320.694,A -85,B 0,C 180,E1 13730.262,E2 13730.262} C_VEL
LIN {X 0,Y 359.419,Z 311.451,A -85,B 0,C 180,E1 13730.033,E2 13730.033} C_VEL
LIN {X 0,Y 348.912,Z 298.266,A -85,B 0,C 180,E1 13727.13,E2 13727.13} C_VEL
LIN {X 0,Y 338.154,Z 285.644,A -85,B 0,C 180,E1 13723.834,E2 13723.834} C_VEL
LIN {X 0,Y 327.65,Z 274.663,A -85,B 0,C 180,E1 13720.198,E2 13720.198} C_VEL
LIN {X 0,Y 321.919,Z 268.875,A -85,B 0,C 180,E1 13717.917,E2 13717.917} C_VEL
LIN {X 0,Y 319.337,Z 264.039,A -85,B 0,C 180,E1 13714.523,E2 13714.523} C_VEL
LIN {X 0,Y 317.198,Z 259.923,A -85,B 0,C 180,E1 13710.918,E2 13710.918} C_VEL
LIN {X 0,Y 316.191,Z 258.597,A -85,B 0,C 180,E1 13709.143,E2 13709.143} C_VEL
LIN {X 0,Y 314.484,Z 254.35,A -85,B 0,C 180,E1 13702.429,E2 13702.429} C_VEL
LIN {X 0,Y 314.252,Z 254.229,A -85,B 0,C 180,E1 13696.45,E2 13696.45} C_VEL
LIN {X 0,Y 314.541,Z 254.843,A -85,B 0,C 180,E1 13694.357,E2 13694.357} C_VEL
LIN {X 0,Y 317.205,Z 259.87,A -85,B 0,C 180,E1 13686.88,E2 13686.88} C_VEL
LIN {X 0,Y 319.765,Z 264.792,A -85,B 0,C 180,E1 13682.689,E2 13682.689} C_VEL
LIN {X 0,Y 322.32,Z 270.018,A -85,B 0,C 180,E1 13679.29,E2 13679.29} C_VEL
LIN {X 0,Y 324.686,Z 274.837,A -85,B 0,C 180,E1 13676.646,E2 13676.646} C_VEL
LIN {X 0,Y 327.133,Z 279.854,A -85,B 0,C 180,E1 13674.212,E2 13674.212} C_VEL
LIN {X 0,Y 330.252,Z 286.125,A -85,B 0,C 180,E1 13671.469,E2 13671.469} C_VEL
LIN {X 0,Y 335.253,Z 297.241,A -85,B 0,C 180,E1 13667.426,E2 13667.426} C_VEL
LIN {X 0,Y 340.641,Z 310.292,A -85,B 0,C 180,E1 13663.459,E2 13663.459} C_VEL
LIN {X 0,Y 346.06,Z 324.677,A -85,B 0,C 180,E1 13659.714,E2 13659.714} C_VEL
LIN {X 0,Y 347.62,Z 329.446,A -85,B 0,C 180,E1 13658.619,E2 13658.619} C_VEL
LIN {X 0,Y 341.615,Z 359.598,A -85,B 0,C 180,E1 13655.35,E2 13655.35} C_VEL
LIN {X 0,Y 339.112,Z 382.33,A -85,B 0,C 180,E1 13652.559,E2 13652.559} C_VEL
LIN {X 0,Y 338.951,Z 403.266,A -85,B 0,C 180,E1 13649.742,E2 13649.742} C_VEL
LIN {X 0,Y 345.125,Z 424.22,A -85,B 0,C 180,E1 13647.616,E2 13647.616} C_VEL
LIN {X 0,Y 352.972,Z 444.505,A -85,B 0,C 180,E1 13645.344,E2 13645.344} C_VEL
LIN {X 0,Y 356.115,Z 451.884,A -85,B 0,C 180,E1 13644.498,E2 13644.498} C_VEL
LIN {X 0,Y 352.219,Z 473.692,A -85,B 0,C 180,E1 13644.384,E2 13644.384} C_VEL
LIN {X 0,Y 348.201,Z 497.274,A -85,B 0,C 180,E1 13643.924,E2 13643.924} C_VEL
LIN {X 0,Y 343.462,Z 526.274,A -85,B 0,C 180,E1 13642.906,E2 13642.906} C_VEL
LIN {X 0,Y 337.783,Z 553.774,A -85,B 0,C 180,E1 13641.667,E2 13641.667} C_VEL
LIN {X 0,Y 331.937,Z 579.287,A -85,B 0,C 180,E1 13640.184,E2 13640.184} C_VEL
LIN {X 0,Y 326.033,Z 603.166,A -85,B 0,C 180,E1 13638.442,E2 13638.442} C_VEL
LIN {X 0,Y 319.844,Z 626.313,A -85,B 0,C 180,E1 13636.36,E2 13636.36} C_VEL
LIN {X 0,Y 314.176,Z 646.022,A -85,B 0,C 180,E1 13634.184,E2 13634.184} C_VEL
LIN {X 0,Y 308.563,Z 663.98,A -85,B 0,C 180,E1 13631.751,E2 13631.751} C_VEL
LIN {X 0,Y 302.749,Z 681.541,A -85,B 0,C 180,E1 13628.865,E2 13628.865} C_VEL
LIN {X 0,Y 297.508,Z 696.937,A -85,B 0,C 180,E1 13625.787,E2 13625.787} C_VEL
LIN {X 0,Y 292.504,Z 711.697,A -85,B 0,C 180,E1 13622.225,E2 13622.225} C_VEL
LIN {X 0,Y 288.43,Z 724.081,A -85,B 0,C 180,E1 13618.58,E2 13618.58} C_VEL
LIN {X 0,Y 284.988,Z 735.554,A -85,B 0,C 180,E1 13614.456,E2 13614.456} C_VEL
LIN {X 0,Y 282.624,Z 744.687,A -85,B 0,C 180,E1 13610.364,E2 13610.364} C_VEL
LIN {X 0,Y 281.134,Z 752.206,A -85,B 0,C 180,E1 13606.105,E2 13606.105} C_VEL
LIN {X 0,Y 280.432,Z 757.791,A -85,B 0,C 180,E1 13601.934,E2 13601.934} C_VEL
LIN {X 0,Y 280.269,Z 761.65,A -85,B 0,C 180,E1 13597.791,E2 13597.791} C_VEL
LIN {X 0,Y 280.337,Z 763.841,A -85,B 0,C 180,E1 13593.885,E2 13593.885} C_VEL
LIN {X 0,Y 280.4,Z 764.618,A -85,B 0,C 180,E1 13590,E2 13590} C_VEL
LIN {X 0,Y 280.323,Z 764.003,A -85,B 0,C 180,E1 13586.114,E2 13586.114} C_VEL
LIN {X 0,Y 280.245,Z 762.009,A -85,B 0,C 180,E1 13582.208,E2 13582.208} C_VEL
LIN {X 0,Y 280.406,Z 758.384,A -85,B 0,C 180,E1 13578.064,E2 13578.064} C_VEL
LIN {X 0,Y 281.172,Z 752.853,A -85,B 0,C 180,E1 13573.684,E2 13573.684} C_VEL
LIN {X 0,Y 282.806,Z 745.529,A -85,B 0,C 180,E1 13569.295,E2 13569.295} C_VEL
LIN {X 0,Y 285.376,Z 736.71,A -85,B 0,C 180,E1 13565.137,E2 13565.137} C_VEL
LIN {X 0,Y 289.257,Z 725.354,A -85,B 0,C 180,E1 13560.831,E2 13560.831} C_VEL
LIN {X 0,Y 293.896,Z 713.019,A -85,B 0,C 180,E1 13557.02,E2 13557.02} C_VEL
LIN {X 0,Y 299.627,Z 698.365,A -85,B 0,C 180,E1 13553.321,E2 13553.321} C_VEL
LIN {X 0,Y 305.891,Z 682.431,A -85,B 0,C 180,E1 13550.024,E2 13550.024} C_VEL
LIN {X 0,Y 312.497,Z 665.211,A -85,B 0,C 180,E1 13547.113,E2 13547.113} C_VEL
LIN {X 0,Y 318.952,Z 647.344,A -85,B 0,C 180,E1 13544.634,E2 13544.634} C_VEL
LIN {X 0,Y 325.58,Z 627.589,A -85,B 0,C 180,E1 13542.406,E2 13542.406} C_VEL
LIN {X 0,Y 331.669,Z 607.225,A -85,B 0,C 180,E1 13540.563,E2 13540.563} C_VEL
LIN {X 0,Y 338.459,Z 582.526,A -85,B 0,C 180,E1 13538.748,E2 13538.748} C_VEL
LIN {X 0,Y 345.057,Z 556.528,A -85,B 0,C 180,E1 13537.244,E2 13537.244} C_VEL
LIN {X 0,Y 351.547,Z 528.473,A -85,B 0,C 180,E1 13535.985,E2 13535.985} C_VEL
LIN {X 0,Y 352.122,Z 525.536,A -85,B 0,C 180,E1 13535.853,E2 13535.853} C_VEL
LIN {X 0,Y 348.948,Z 530.786,A -85,B 0,C 180,E1 13535.567,E2 13535.567} C_VEL
LIN {X 0,Y 343.46,Z 540.754,A -85,B 0,C 180,E1 13535.197,E2 13535.197} C_VEL
LIN {X 0,Y 338.389,Z 548.257,A -85,B 0,C 180,E1 13534.701,E2 13534.701} C_VEL
LIN {X 0,Y 333.451,Z 556.159,A -85,B 0,C 180,E1 13534.313,E2 13534.313} C_VEL
LIN {X 0,Y 328.552,Z 562.455,A -85,B 0,C 180,E1 13533.737,E2 13533.737} C_VEL
LIN {X 0,Y 323.668,Z 569.209,A -85,B 0,C 180,E1 13533.251,E2 13533.251} C_VEL
LIN {X 0,Y 319.505,Z 573.773,A -85,B 0,C 180,E1 13532.668,E2 13532.668} C_VEL
LIN {X 0,Y 315.373,Z 579.071,A -85,B 0,C 180,E1 13532.183,E2 13532.183} C_VEL
LIN {X 0,Y 311.726,Z 582.821,A -85,B 0,C 180,E1 13531.521,E2 13531.521} C_VEL
LIN {X 0,Y 308.548,Z 599.372,A -85,B 0,C 180,E1 13529.719,E2 13529.719} C_VEL
LIN {X 0,Y 305.114,Z 614.601,A -85,B 0,C 180,E1 13527.625,E2 13527.625} C_VEL
LIN {X 0,Y 301.629,Z 627.879,A -85,B 0,C 180,E1 13525.316,E2 13525.316} C_VEL
LIN {X 0,Y 298.332,Z 639.111,A -85,B 0,C 180,E1 13522.878,E2 13522.878} C_VEL
LIN {X 0,Y 294.924,Z 649.375,A -85,B 0,C 180,E1 13520.023,E2 13520.023} C_VEL
LIN {X 0,Y 291.978,Z 657.302,A -85,B 0,C 180,E1 13517.127,E2 13517.127} C_VEL
LIN {X 0,Y 289.497,Z 663.205,A -85,B 0,C 180,E1 13514.194,E2 13514.194} C_VEL
LIN {X 0,Y 287.363,Z 667.616,A -85,B 0,C 180,E1 13511.032,E2 13511.032} C_VEL
LIN {X 0,Y 285.703,Z 670.127,A -85,B 0,C 180,E1 13507.844,E2 13507.844} C_VEL
LIN {X 0,Y 284.514,Z 670.891,A -85,B 0,C 180,E1 13504.635,E2 13504.635} C_VEL
LIN {X 0,Y 283.734,Z 669.941,A -85,B 0,C 180,E1 13501.413,E2 13501.413} C_VEL
LIN {X 0,Y 283.316,Z 667.3,A -85,B 0,C 180,E1 13498.179,E2 13498.179} C_VEL
LIN {X 0,Y 283.223,Z 662.855,A -85,B 0,C 180,E1 13494.936,E2 13494.936} C_VEL
LIN {X 0,Y 283.486,Z 656.579,A -85,B 0,C 180,E1 13491.685,E2 13491.685} C_VEL
LIN {X 0,Y 284.092,Z 648.805,A -85,B 0,C 180,E1 13488.632,E2 13488.632} C_VEL
LIN {X 0,Y 285.056,Z 638.887,A -85,B 0,C 180,E1 13485.579,E2 13485.579} C_VEL
LIN {X 0,Y 286.338,Z 627.407,A -85,B 0,C 180,E1 13482.733,E2 13482.733} C_VEL
LIN {X 0,Y 287.133,Z 620.543,A -85,B 0,C 180,E1 13481.293,E2 13481.293} C_VEL
LIN {X 0,Y 288.596,Z 621.037,A -85,B 0,C 180,E1 13480.573,E2 13480.573} C_VEL
LIN {X 0,Y 292.152,Z 620.088,A -85,B 0,C 180,E1 13479.568,E2 13479.568} C_VEL
LIN {X 0,Y 295.418,Z 619.645,A -85,B 0,C 180,E1 13478.559,E2 13478.559} C_VEL
LIN {X 0,Y 297.489,Z 618.96,A -85,B 0,C 180,E1 13478.07,E2 13478.07} C_VEL
LIN {X 0,Y 301.637,Z 618.198,A -85,B 0,C 180,E1 13476.974,E2 13476.974} C_VEL
LIN {X 0,Y 304.675,Z 617.346,A -85,B 0,C 180,E1 13476.292,E2 13476.292} C_VEL
LIN {X 0,Y 309.926,Z 615.83,A -85,B 0,C 180,E1 13475.203,E2 13475.203} C_VEL
LIN {X 0,Y 317.257,Z 613.586,A -85,B 0,C 180,E1 13473.818,E2 13473.818} C_VEL
LIN {X 0,Y 326.23,Z 610.568,A -85,B 0,C 180,E1 13472.345,E2 13472.345} C_VEL
LIN {X 0,Y 319.58,Z 627.608,A -85,B 0,C 180,E1 13469.91,E2 13469.91} C_VEL
LIN {X 0,Y 312.922,Z 643.229,A -85,B 0,C 180,E1 13467.178,E2 13467.178} C_VEL
LIN {X 0,Y 306.281,Z 657.8,A -85,B 0,C 180,E1 13464.058,E2 13464.058} C_VEL
LIN {X 0,Y 300.085,Z 670.895,A -85,B 0,C 180,E1 13460.625,E2 13460.625} C_VEL
LIN {X 0,Y 294.678,Z 682.157,A -85,B 0,C 180,E1 13456.999,E2 13456.999} C_VEL
LIN {X 0,Y 290.001,Z 692.147,A -85,B 0,C 180,E1 13453.035,E2 13453.035} C_VEL
LIN {X 0,Y 286.175,Z 700.806,A -85,B 0,C 180,E1 13448.712,E2 13448.712} C_VEL
LIN {X 0,Y 283.499,Z 707.576,A -85,B 0,C 180,E1 13444.354,E2 13444.354} C_VEL
LIN {X 0,Y 281.819,Z 712.63,A -85,B 0,C 180,E1 13440.017,E2 13440.017} C_VEL
LIN {X 0,Y 280.915,Z 715.999,A -85,B 0,C 180,E1 13435.737,E2 13435.737} C_VEL
LIN {X 0,Y 280.516,Z 717.923,A -85,B 0,C 180,E1 13431.517,E2 13431.517} C_VEL
LIN {X 0,Y 280.4,Z 718.521,A -85,B 0,C 180,E1 13427.43,E2 13427.43} C_VEL
LIN {X 0,Y 280.439,Z 717.714,A -85,B 0,C 180,E1 13423.4,E2 13423.4} C_VEL
LIN {X 0,Y 280.671,Z 715.557,A -85,B 0,C 180,E1 13419.225,E2 13419.225} C_VEL
LIN {X 0,Y 281.315,Z 712.071,A -85,B 0,C 180,E1 13415.098,E2 13415.098} C_VEL
LIN {X 0,Y 282.605,Z 706.789,A -85,B 0,C 180,E1 13410.811,E2 13410.811} C_VEL
LIN {X 0,Y 284.712,Z 699.879,A -85,B 0,C 180,E1 13406.578,E2 13406.578} C_VEL
LIN {X 0,Y 287.764,Z 691.223,A -85,B 0,C 180,E1 13402.413,E2 13402.413} C_VEL
LIN {X 0,Y 291.619,Z 681.175,A -85,B 0,C 180,E1 13398.53,E2 13398.53} C_VEL
LIN {X 0,Y 296.142,Z 669.786,A -85,B 0,C 180,E1 13394.932,E2 13394.932} C_VEL
LIN {X 0,Y 301.516,Z 656.256,A -85,B 0,C 180,E1 13391.437,E2 13391.437} C_VEL
LIN {X 0,Y 307.374,Z 641.069,A -85,B 0,C 180,E1 13388.233,E2 13388.233} C_VEL
LIN {X 0,Y 312.549,Z 626.774,A -85,B 0,C 180,E1 13385.743,E2 13385.743} C_VEL
LIN {X 0,Y 313.714,Z 621.298,A -85,B 0,C 180,E1 13384.762,E2 13384.762} C_VEL
LIN {X 0,Y 313.823,Z 607.477,A -85,B 0,C 180,E1 13382.089,E2 13382.089} C_VEL
LIN {X 0,Y 314.979,Z 601.465,A -85,B 0,C 180,E1 13381.219,E2 13381.219} C_VEL
LIN {X 0,Y 320.406,Z 583.149,A -85,B 0,C 180,E1 13379.218,E2 13379.218} C_VEL
LIN {X 0,Y 325.212,Z 564.48,A -85,B 0,C 180,E1 13377.555,E2 13377.555} C_VEL
LIN {X 0,Y 329.424,Z 544.94,A -85,B 0,C 180,E1 13376.15,E2 13376.15} C_VEL
LIN {X 0,Y 333.044,Z 523.657,A -85,B 0,C 180,E1 13374.965,E2 13374.965} C_VEL
LIN {X 0,Y 335.632,Z 502.299,A -85,B 0,C 180,E1 13374.085,E2 13374.085} C_VEL
LIN {X 0,Y 341.253,Z 449.903,A -85,B 0,C 180,E1 13372.485,E2 13372.485} C_VEL
LIN {X 0,Y 349.568,Z 370.349,A -85,B 0,C 180,E1 13370.396,E2 13370.396} C_VEL
LIN {X 0,Y 354.29,Z 315.801,A -85,B 0,C 180,E1 13369.088,E2 13369.088} C_VEL
LIN {X 0,Y 343.919,Z 302.655,A -85,B 0,C 180,E1 13366.078,E2 13366.078} C_VEL
LIN {X 0,Y 334.279,Z 291.581,A -85,B 0,C 180,E1 13362.999,E2 13362.999} C_VEL
LIN {X 0,Y 328.064,Z 284.977,A -85,B 0,C 180,E1 13360.825,E2 13360.825} C_VEL
LIN {X 0,Y 324.132,Z 280.922,A -85,B 0,C 180,E1 13359.34,E2 13359.34} C_VEL
LIN {X 0,Y 318.965,Z 275.773,A -85,B 0,C 180,E1 13357.229,E2 13357.229} C_VEL
LIN {X 0,Y 316.212,Z 273.181,A -85,B 0,C 180,E1 13355.956,E2 13355.956} C_VEL
LIN {X 0,Y 315.049,Z 270.662,A -85,B 0,C 180,E1 13354.177,E2 13354.177} C_VEL
LIN {X 0,Y 313.084,Z 266.459,A -85,B 0,C 180,E1 13350.517,E2 13350.517} C_VEL
LIN {X 0,Y 310.598,Z 261.344,A -85,B 0,C 180,E1 13342.498,E2 13342.498} C_VEL
LIN {X 0,Y 310.354,Z 261.215,A -85,B 0,C 180,E1 13336.47,E2 13336.47} C_VEL
LIN {X 0,Y 310.623,Z 261.866,A -85,B 0,C 180,E1 13334.331,E2 13334.331} C_VEL
LIN {X 0,Y 313.108,Z 266.574,A -85,B 0,C 180,E1 13327.155,E2 13327.155} C_VEL
LIN {X 0,Y 315.662,Z 271.809,A -85,B 0,C 180,E1 13322.724,E2 13322.724} C_VEL
LIN {X 0,Y 317.962,Z 276.496,A -85,B 0,C 180,E1 13319.602,E2 13319.602} C_VEL
LIN {X 0,Y 320.221,Z 281.24,A -85,B 0,C 180,E1 13316.958,E2 13316.958} C_VEL
LIN {X 0,Y 322.791,Z 286.644,A -85,B 0,C 180,E1 13314.312,E2 13314.312} C_VEL
LIN {X 0,Y 326.013,Z 293.475,A -85,B 0,C 180,E1 13311.357,E2 13311.357} C_VEL
LIN {X 0,Y 330.344,Z 303.242,A -85,B 0,C 180,E1 13307.769,E2 13307.769} C_VEL
LIN {X 0,Y 335.369,Z 315.731,A -85,B 0,C 180,E1 13303.903,E2 13303.903} C_VEL
LIN {X 0,Y 340.664,Z 330.123,A -85,B 0,C 180,E1 13300.095,E2 13300.095} C_VEL
LIN {X 0,Y 341.65,Z 333.603,A -85,B 0,C 180,E1 13299.306,E2 13299.306} C_VEL
LIN {X 0,Y 335.685,Z 362.693,A -85,B 0,C 180,E1 13296.104,E2 13296.104} C_VEL
LIN {X 0,Y 333.002,Z 385.709,A -85,B 0,C 180,E1 13293.232,E2 13293.232} C_VEL
LIN {X 0,Y 332.646,Z 399.399,A -85,B 0,C 180,E1 13291.414,E2 13291.414} C_VEL
LIN {X 0,Y 338.224,Z 420.951,A -85,B 0,C 180,E1 13289.267,E2 13289.267} C_VEL
LIN {X 0,Y 345.606,Z 442.379,A -85,B 0,C 180,E1 13286.903,E2 13286.903} C_VEL
LIN {X 0,Y 350.456,Z 454.386,A -85,B 0,C 180,E1 13285.5,E2 13285.5} C_VEL
LIN {X 0,Y 346.524,Z 476.173,A -85,B 0,C 180,E1 13285.339,E2 13285.339} C_VEL
LIN {X 0,Y 342.637,Z 498.349,A -85,B 0,C 180,E1 13284.875,E2 13284.875} C_VEL
LIN {X 0,Y 337.916,Z 526.023,A -85,B 0,C 180,E1 13283.879,E2 13283.879} C_VEL
LIN {X 0,Y 331.792,Z 554.807,A -85,B 0,C 180,E1 13282.566,E2 13282.566} C_VEL
LIN {X 0,Y 325.816,Z 580.102,A -85,B 0,C 180,E1 13281.072,E2 13281.072} C_VEL
LIN {X 0,Y 319.483,Z 604.74,A -85,B 0,C 180,E1 13279.232,E2 13279.232} C_VEL
LIN {X 0,Y 312.904,Z 628.67,A -85,B 0,C 180,E1 13277.033,E2 13277.033} C_VEL
LIN {X 0,Y 307.053,Z 647.878,A -85,B 0,C 180,E1 13274.815,E2 13274.815} C_VEL
LIN {X 0,Y 300.985,Z 666.451,A -85,B 0,C 180,E1 13272.202,E2 13272.202} C_VEL
LIN {X 0,Y 295.146,Z 683.236,A -85,B 0,C 180,E1 13269.308,E2 13269.308} C_VEL
LIN {X 0,Y 289.454,Z 699.247,A -85,B 0,C 180,E1 13265.96,E2 13265.96} C_VEL
LIN {X 0,Y 284.637,Z 712.762,A -85,B 0,C 180,E1 13262.51,E2 13262.51} C_VEL
LIN {X 0,Y 280.273,Z 725.541,A -85,B 0,C 180,E1 13258.557,E2 13258.557} C_VEL
LIN {X 0,Y 276.963,Z 736.129,A -85,B 0,C 180,E1 13254.529,E2 13254.529} C_VEL
LIN {X 0,Y 274.444,Z 745.596,A -85,B 0,C 180,E1 13250.027,E2 13250.027} C_VEL
LIN {X 0,Y 273.031,Z 752.643,A -85,B 0,C 180,E1 13245.723,E2 13245.723} C_VEL
LIN {X 0,Y 272.385,Z 758.129,A -85,B 0,C 180,E1 13241.218,E2 13241.218} C_VEL
LIN {X 0,Y 272.298,Z 761.674,A -85,B 0,C 180,E1 13236.96,E2 13236.96} C_VEL
LIN {X 0,Y 272.384,Z 763.524,A -85,B 0,C 180,E1 13232.945,E2 13232.945} C_VEL
LIN {X 0,Y 272.411,Z 763.966,A -85,B 0,C 180,E1 13229.158,E2 13229.158} C_VEL
LIN {X 0,Y 272.326,Z 763.158,A -85,B 0,C 180,E1 13225.367,E2 13225.367} C_VEL
LIN {X 0,Y 272.254,Z 760.943,A -85,B 0,C 180,E1 13221.339,E2 13221.339} C_VEL
LIN {X 0,Y 272.516,Z 757.09,A -85,B 0,C 180,E1 13217.067,E2 13217.067} C_VEL
LIN {X 0,Y 273.483,Z 751.363,A -85,B 0,C 180,E1 13212.554,E2 13212.554} C_VEL
LIN {X 0,Y 275.436,Z 743.796,A -85,B 0,C 180,E1 13208.043,E2 13208.043} C_VEL
LIN {X 0,Y 278.545,Z 734.23,A -85,B 0,C 180,E1 13203.569,E2 13203.569} C_VEL
LIN {X 0,Y 282.722,Z 723.116,A -85,B 0,C 180,E1 13199.385,E2 13199.385} C_VEL
LIN {X 0,Y 287.832,Z 710.497,A -85,B 0,C 180,E1 13195.512,E2 13195.512} C_VEL
LIN {X 0,Y 293.71,Z 696.367,A -85,B 0,C 180,E1 13191.963,E2 13191.963} C_VEL
LIN {X 0,Y 300.207,Z 680.81,A -85,B 0,C 180,E1 13188.741,E2 13188.741} C_VEL
LIN {X 0,Y 306.894,Z 664.189,A -85,B 0,C 180,E1 13185.924,E2 13185.924} C_VEL
LIN {X 0,Y 314.022,Z 645.361,A -85,B 0,C 180,E1 13183.318,E2 13183.318} C_VEL
LIN {X 0,Y 320.775,Z 625.973,A -85,B 0,C 180,E1 13181.156,E2 13181.156} C_VEL
LIN {X 0,Y 326.772,Z 606.572,A -85,B 0,C 180,E1 13179.411,E2 13179.411} C_VEL
LIN {X 0,Y 333.799,Z 581.752,A -85,B 0,C 180,E1 13177.6,E2 13177.6} C_VEL
LIN {X 0,Y 340.801,Z 555.038,A -85,B 0,C 180,E1 13176.072,E2 13176.072} C_VEL
LIN {X 0,Y 341.69,Z 551.066,A -85,B 0,C 180,E1 13175.848,E2 13175.848} C_VEL
LIN {X 0,Y 335.646,Z 560.441,A -85,B 0,C 180,E1 13175.408,E2 13175.408} C_VEL
LIN {X 0,Y 330.112,Z 567.424,A -85,B 0,C 180,E1 13174.833,E2 13174.833} C_VEL
LIN {X 0,Y 324.712,Z 574.535,A -85,B 0,C 180,E1 13174.297,E2 13174.297} C_VEL
LIN {X 0,Y 320.887,Z 578.692,A -85,B 0,C 180,E1 13173.792,E2 13173.792} C_VEL
LIN {X 0,Y 315.789,Z 584.737,A -85,B 0,C 180,E1 13173.213,E2 13173.213} C_VEL
LIN {X 0,Y 312.433,Z 587.857,A -85,B 0,C 180,E1 13172.683,E2 13172.683} C_VEL
LIN {X 0,Y 308.157,Z 592.729,A -85,B 0,C 180,E1 13172.128,E2 13172.128} C_VEL
LIN {X 0,Y 304.466,Z 596.187,A -85,B 0,C 180,E1 13171.415,E2 13171.415} C_VEL
LIN {X 0,Y 300.882,Z 611.193,A -85,B 0,C 180,E1 13169.459,E2 13169.459} C_VEL
LIN {X 0,Y 297.123,Z 624.792,A -85,B 0,C 180,E1 13167.235,E2 13167.235} C_VEL
LIN {X 0,Y 293.398,Z 636.827,A -85,B 0,C 180,E1 13164.781,E2 13164.781} C_VEL
LIN {X 0,Y 289.759,Z 647.207,A -85,B 0,C 180,E1 13162.093,E2 13162.093} C_VEL
LIN {X 0,Y 286.343,Z 655.993,A -85,B 0,C 180,E1 13159.161,E2 13159.161} C_VEL
LIN {X 0,Y 283.406,Z 662.628,A -85,B 0,C 180,E1 13156.183,E2 13156.183} C_VEL
LIN {X 0,Y 280.99,Z 667.494,A -85,B 0,C 180,E1 13153.163,E2 13153.163} C_VEL
LIN {X 0,Y 278.911,Z 670.825,A -85,B 0,C 180,E1 13149.908,E2 13149.908} C_VEL
LIN {X 0,Y 277.351,Z 672.334,A -85,B 0,C 180,E1 13146.624,E2 13146.624} C_VEL
LIN {X 0,Y 276.273,Z 672.147,A -85,B 0,C 180,E1 13143.319,E2 13143.319} C_VEL
LIN {X 0,Y 275.614,Z 670.262,A -85,B 0,C 180,E1 13139.999,E2 13139.999} C_VEL
LIN {X 0,Y 275.307,Z 666.615,A -85,B 0,C 180,E1 13136.668,E2 13136.668} C_VEL
LIN {X 0,Y 275.372,Z 661.159,A -85,B 0,C 180,E1 13133.327,E2 13133.327} C_VEL
LIN {X 0,Y 275.792,Z 654.288,A -85,B 0,C 180,E1 13130.189,E2 13130.189} C_VEL
LIN {X 0,Y 276.586,Z 645.423,A -85,B 0,C 180,E1 13127.048,E2 13127.048} C_VEL
LIN {X 0,Y 277.752,Z 634.567,A -85,B 0,C 180,E1 13123.979,E2 13123.979} C_VEL
LIN {X 0,Y 278.636,Z 627.522,A -85,B 0,C 180,E1 13122.24,E2 13122.24} C_VEL
LIN {X 0,Y 280.117,Z 627.918,A -85,B 0,C 180,E1 13121.477,E2 13121.477} C_VEL
LIN {X 0,Y 283.236,Z 627.24,A -85,B 0,C 180,E1 13120.484,E2 13120.484} C_VEL
LIN {X 0,Y 286.578,Z 626.852,A -85,B 0,C 180,E1 13119.366,E2 13119.366} C_VEL
LIN {X 0,Y 288.409,Z 626.38,A -85,B 0,C 180,E1 13118.865,E2 13118.865} C_VEL
LIN {X 0,Y 292.475,Z 625.643,A -85,B 0,C 180,E1 13117.699,E2 13117.699} C_VEL
LIN {X 0,Y 299.574,Z 623.985,A -85,B 0,C 180,E1 13115.971,E2 13115.971} C_VEL
LIN {X 0,Y 306.524,Z 622.166,A -85,B 0,C 180,E1 13114.495,E2 13114.495} C_VEL
LIN {X 0,Y 315.6,Z 619.358,A -85,B 0,C 180,E1 13112.856,E2 13112.856} C_VEL
LIN {X 0,Y 318.06,Z 618.621,A -85,B 0,C 180,E1 13112.438,E2 13112.438} C_VEL
LIN {X 0,Y 311.253,Z 634.66,A -85,B 0,C 180,E1 13109.925,E2 13109.925} C_VEL
LIN {X 0,Y 304.381,Z 649.619,A -85,B 0,C 180,E1 13107.066,E2 13107.066} C_VEL
LIN {X 0,Y 297.512,Z 663.739,A -85,B 0,C 180,E1 13103.763,E2 13103.763} C_VEL
LIN {X 0,Y 291.35,Z 675.979,A -85,B 0,C 180,E1 13100.24,E2 13100.24} C_VEL
LIN {X 0,Y 285.854,Z 686.862,A -85,B 0,C 180,E1 13096.39,E2 13096.39} C_VEL
LIN {X 0,Y 281.207,Z 696.309,A -85,B 0,C 180,E1 13092.223,E2 13092.223} C_VEL
LIN {X 0,Y 277.552,Z 704.277,A -85,B 0,C 180,E1 13087.765,E2 13087.765} C_VEL
LIN {X 0,Y 274.956,Z 710.642,A -85,B 0,C 180,E1 13083.057,E2 13083.057} C_VEL
LIN {X 0,Y 273.446,Z 715.102,A -85,B 0,C 180,E1 13078.382,E2 13078.382} C_VEL
LIN {X 0,Y 272.74,Z 717.761,A -85,B 0,C 180,E1 13074.012,E2 13074.012} C_VEL
LIN {X 0,Y 272.473,Z 719.038,A -85,B 0,C 180,E1 13069.731,E2 13069.731} C_VEL
LIN {X 0,Y 272.425,Z 718.976,A -85,B 0,C 180,E1 13065.76,E2 13065.76} C_VEL
LIN {X 0,Y 272.539,Z 717.548,A -85,B 0,C 180,E1 13061.427,E2 13061.427} C_VEL
LIN {X 0,Y 272.958,Z 714.793,A -85,B 0,C 180,E1 13057.155,E2 13057.155} C_VEL
LIN {X 0,Y 273.958,Z 710.364,A -85,B 0,C 180,E1 13052.72,E2 13052.72} C_VEL
LIN {X 0,Y 275.745,Z 704.299,A -85,B 0,C 180,E1 13048.338,E2 13048.338} C_VEL
LIN {X 0,Y 278.445,Z 696.545,A -85,B 0,C 180,E1 13044.023,E2 13044.023} C_VEL
LIN {X 0,Y 282.18,Z 686.945,A -85,B 0,C 180,E1 13039.796,E2 13039.796} C_VEL
LIN {X 0,Y 286.485,Z 676.499,A -85,B 0,C 180,E1 13036.066,E2 13036.066} C_VEL
LIN {X 0,Y 291.662,Z 664.099,A -85,B 0,C 180,E1 13032.442,E2 13032.442} C_VEL
LIN {X 0,Y 297.356,Z 650.168,A -85,B 0,C 180,E1 13029.119,E2 13029.119} C_VEL
LIN {X 0,Y 303.403,Z 634.674,A -85,B 0,C 180,E1 13026.088,E2 13026.088} C_VEL
LIN {X 0,Y 309.261,Z 618.621,A -85,B 0,C 180,E1 13023.503,E2 13023.503} C_VEL
LIN {X 0,Y 314.979,Z 601.465,A -85,B 0,C 180,E1 13021.219,E2 13021.219} C_VEL
LIN {X 0,Y 316.175,Z 595.364,A -85,B 0,C 180,E1 13020.376,E2 13020.376} C_VEL
LIN {X 0,Y 316.34,Z 580.024,A -85,B 0,C 180,E1 13018.015,E2 13018.015} C_VEL
LIN {X 0,Y 317.331,Z 573.493,A -85,B 0,C 180,E1 13017.283,E2 13017.283} C_VEL
LIN {X 0,Y 322.085,Z 553.639,A -85,B 0,C 180,E1 13015.706,E2 13015.706} C_VEL
LIN {X 0,Y 325.96,Z 533.702,A -85,B 0,C 180,E1 13014.46,E2 13014.46} C_VEL
LIN {X 0,Y 328.991,Z 513.213,A -85,B 0,C 180,E1 13013.473,E2 13013.473} C_VEL
LIN {X 0,Y 333.51,Z 472.103,A -85,B 0,C 180,E1 13012.085,E2 13012.085} C_VEL
LIN {X 0,Y 342.484,Z 392.677,A -85,B 0,C 180,E1 13009.896,E2 13009.896} C_VEL
LIN {X 0,Y 349.155,Z 323.181,A -85,B 0,C 180,E1 13008.219,E2 13008.219} C_VEL
LIN {X 0,Y 349.347,Z 320.298,A -85,B 0,C 180,E1 13008.142,E2 13008.142} C_VEL
LIN {X 0,Y 339.884,Z 308.271,A -85,B 0,C 180,E1 13005.271,E2 13005.271} C_VEL
LIN {X 0,Y 331.162,Z 298.161,A -85,B 0,C 180,E1 13002.381,E2 13002.381} C_VEL
LIN {X 0,Y 325.387,Z 291.936,A -85,B 0,C 180,E1 13000.304,E2 13000.304} C_VEL
LIN {X 0,Y 321.115,Z 287.488,A -85,B 0,C 180,E1 12998.632,E2 12998.632} C_VEL
LIN {X 0,Y 316.865,Z 283.201,A -85,B 0,C 180,E1 12996.838,E2 12996.838} C_VEL
LIN {X 0,Y 310.933,Z 277.474,A -85,B 0,C 180,E1 12994.024,E2 12994.024} C_VEL
LIN {X 0,Y 308.779,Z 273,A -85,B 0,C 180,E1 12989.913,E2 12989.913} C_VEL
LIN {X 0,Y 306.678,Z 268.316,A -85,B 0,C 180,E1 12982.425,E2 12982.425} C_VEL
LIN {X 0,Y 306.486,Z 268.231,A -85,B 0,C 180,E1 12976.294,E2 12976.294} C_VEL
LIN {X 0,Y 306.702,Z 268.867,A -85,B 0,C 180,E1 12974.346,E2 12974.346} C_VEL
LIN {X 0,Y 309.065,Z 273.524,A -85,B 0,C 180,E1 12967.249,E2 12967.249} C_VEL
LIN {X 0,Y 311.466,Z 278.522,A -85,B 0,C 180,E1 12962.945,E2 12962.945} C_VEL
LIN {X 0,Y 313.803,Z 283.49,A -85,B 0,C 180,E1 12959.635,E2 12959.635} C_VEL
LIN {X 0,Y 315.914,Z 288.002,A -85,B 0,C 180,E1 12957.098,E2 12957.098} C_VEL
LIN {X 0,Y 319.228,Z 294.858,A -85,B 0,C 180,E1 12953.707,E2 12953.707} C_VEL
LIN {X 0,Y 323.813,Z 305.336,A -85,B 0,C 180,E1 12949.504,E2 12949.504} C_VEL
LIN {X 0,Y 328.361,Z 316.643,A -85,B 0,C 180,E1 12945.722,E2 12945.722} C_VEL
LIN {X 0,Y 333.176,Z 329.542,A -85,B 0,C 180,E1 12942.048,E2 12942.048} C_VEL
LIN {X 0,Y 335.85,Z 337.274,A -85,B 0,C 180,E1 12940.07,E2 12940.07} C_VEL
LIN {X 0,Y 329.81,Z 365.777,A -85,B 0,C 180,E1 12936.885,E2 12936.885} C_VEL
LIN {X 0,Y 326.892,Z 389.533,A -85,B 0,C 180,E1 12933.868,E2 12933.868} C_VEL
LIN {X 0,Y 326.719,Z 395.278,A -85,B 0,C 180,E1 12933.131,E2 12933.131} C_VEL
LIN {X 0,Y 331.575,Z 417.026,A -85,B 0,C 180,E1 12931.005,E2 12931.005} C_VEL
LIN {X 0,Y 338.288,Z 439.101,A -85,B 0,C 180,E1 12928.606,E2 12928.606} C_VEL
LIN {X 0,Y 344.835,Z 456.986,A -85,B 0,C 180,E1 12926.518,E2 12926.518} C_VEL
LIN {X 0,Y 340.805,Z 479.036,A -85,B 0,C 180,E1 12926.306,E2 12926.306} C_VEL
LIN {X 0,Y 336.927,Z 500.644,A -85,B 0,C 180,E1 12925.813,E2 12925.813} C_VEL
LIN {X 0,Y 331.306,Z 531.556,A -85,B 0,C 180,E1 12924.646,E2 12924.646} C_VEL
LIN {X 0,Y 325.252,Z 558.521,A -85,B 0,C 180,E1 12923.354,E2 12923.354} C_VEL
LIN {X 0,Y 318.611,Z 585.383,A -85,B 0,C 180,E1 12921.678,E2 12921.678} C_VEL
LIN {X 0,Y 312.189,Z 609.368,A -85,B 0,C 180,E1 12919.805,E2 12919.805} C_VEL
LIN {X 0,Y 305.994,Z 630.753,A -85,B 0,C 180,E1 12917.74,E2 12917.74} C_VEL
LIN {X 0,Y 299.791,Z 650.36,A -85,B 0,C 180,E1 12915.403,E2 12915.403} C_VEL
LIN {X 0,Y 293.658,Z 668.111,A -85,B 0,C 180,E1 12912.786,E2 12912.786} C_VEL
LIN {X 0,Y 287.561,Z 684.918,A -85,B 0,C 180,E1 12909.775,E2 12909.775} C_VEL
LIN {X 0,Y 282.034,Z 699.692,A -85,B 0,C 180,E1 12906.554,E2 12906.554} C_VEL
LIN {X 0,Y 276.779,Z 713.826,A -85,B 0,C 180,E1 12902.811,E2 12902.811} C_VEL
LIN {X 0,Y 272.517,Z 725.729,A -85,B 0,C 180,E1 12898.967,E2 12898.967} C_VEL
LIN {X 0,Y 268.935,Z 736.644,A -85,B 0,C 180,E1 12894.607,E2 12894.607} C_VEL
LIN {X 0,Y 266.483,Z 745.52,A -85,B 0,C 180,E1 12890.193,E2 12890.193} C_VEL
LIN {X 0,Y 265.035,Z 752.422,A -85,B 0,C 180,E1 12885.761,E2 12885.761} C_VEL
LIN {X 0,Y 264.404,Z 757.586,A -85,B 0,C 180,E1 12881.34,E2 12881.34} C_VEL
LIN {X 0,Y 264.318,Z 761.093,A -85,B 0,C 180,E1 12876.952,E2 12876.952} C_VEL
LIN {X 0,Y 264.415,Z 762.889,A -85,B 0,C 180,E1 12872.817,E2 12872.817} C_VEL
LIN {X 0,Y 264.436,Z 763.29,A -85,B 0,C 180,E1 12868.916,E2 12868.916} C_VEL
LIN {X 0,Y 264.337,Z 762.436,A -85,B 0,C 180,E1 12865.009,E2 12865.009} C_VEL
LIN {X 0,Y 264.272,Z 760.171,A -85,B 0,C 180,E1 12860.856,E2 12860.856} C_VEL
LIN {X 0,Y 264.598,Z 756.277,A -85,B 0,C 180,E1 12856.45,E2 12856.45} C_VEL
LIN {X 0,Y 265.795,Z 750.171,A -85,B 0,C 180,E1 12851.579,E2 12851.579} C_VEL
LIN {X 0,Y 268.026,Z 742.455,A -85,B 0,C 180,E1 12846.939,E2 12846.939} C_VEL
LIN {X 0,Y 271.501,Z 732.735,A -85,B 0,C 180,E1 12842.353,E2 12842.353} C_VEL
LIN {X 0,Y 276.096,Z 721.502,A -85,B 0,C 180,E1 12838.08,E2 12838.08} C_VEL
LIN {X 0,Y 281.65,Z 708.698,A -85,B 0,C 180,E1 12834.143,E2 12834.143} C_VEL
LIN {X 0,Y 287.989,Z 694.435,A -85,B 0,C 180,E1 12830.553,E2 12830.553} C_VEL
LIN {X 0,Y 295.134,Z 678.17,A -85,B 0,C 180,E1 12827.214,E2 12827.214} C_VEL
LIN {X 0,Y 302.489,Z 660.665,A -85,B 0,C 180,E1 12824.305,E2 12824.305} C_VEL
LIN {X 0,Y 309.805,Z 641.974,A -85,B 0,C 180,E1 12821.795,E2 12821.795} C_VEL
LIN {X 0,Y 316.598,Z 623.054,A -85,B 0,C 180,E1 12819.735,E2 12819.735} C_VEL
LIN {X 0,Y 323.191,Z 602.164,A -85,B 0,C 180,E1 12817.917,E2 12817.917} C_VEL
LIN {X 0,Y 330.569,Z 576.552,A -85,B 0,C 180,E1 12816.139,E2 12816.139} C_VEL
LIN {X 0,Y 331.64,Z 572.555,A -85,B 0,C 180,E1 12815.901,E2 12815.901} C_VEL
LIN {X 0,Y 325.806,Z 579.802,A -85,B 0,C 180,E1 12815.343,E2 12815.343} C_VEL
LIN {X 0,Y 321.698,Z 584.256,A -85,B 0,C 180,E1 12814.862,E2 12814.862} C_VEL
LIN {X 0,Y 316.275,Z 590.381,A -85,B 0,C 180,E1 12814.244,E2 12814.244} C_VEL
LIN {X 0,Y 312.544,Z 594.031,A -85,B 0,C 180,E1 12813.719,E2 12813.719} C_VEL
LIN {X 0,Y 306.898,Z 599.697,A -85,B 0,C 180,E1 12812.961,E2 12812.961} C_VEL
LIN {X 0,Y 303.744,Z 602.501,A -85,B 0,C 180,E1 12812.449,E2 12812.449} C_VEL
LIN {X 0,Y 299.637,Z 606.329,A -85,B 0,C 180,E1 12811.818,E2 12811.818} C_VEL
LIN {X 0,Y 297.067,Z 608.344,A -85,B 0,C 180,E1 12811.276,E2 12811.276} C_VEL
LIN {X 0,Y 292.765,Z 622.818,A -85,B 0,C 180,E1 12809.009,E2 12809.009} C_VEL
LIN {X 0,Y 288.896,Z 634.502,A -85,B 0,C 180,E1 12806.738,E2 12806.738} C_VEL
LIN {X 0,Y 284.783,Z 645.598,A -85,B 0,C 180,E1 12804.033,E2 12804.033} C_VEL
LIN {X 0,Y 281.12,Z 654.487,A -85,B 0,C 180,E1 12801.271,E2 12801.271} C_VEL
LIN {X 0,Y 277.691,Z 661.868,A -85,B 0,C 180,E1 12798.255,E2 12798.255} C_VEL
LIN {X 0,Y 274.814,Z 667.408,A -85,B 0,C 180,E1 12795.186,E2 12795.186} C_VEL
LIN {X 0,Y 272.303,Z 671.404,A -85,B 0,C 180,E1 12791.865,E2 12791.865} C_VEL
LIN {X 0,Y 270.344,Z 673.55,A -85,B 0,C 180,E1 12788.507,E2 12788.507} C_VEL
LIN {X 0,Y 268.94,Z 674.018,A -85,B 0,C 180,E1 12785.118,E2 12785.118} C_VEL
LIN {X 0,Y 268.013,Z 672.768,A -85,B 0,C 180,E1 12781.71,E2 12781.71} C_VEL
LIN {X 0,Y 267.495,Z 669.76,A -85,B 0,C 180,E1 12778.286,E2 12778.286} C_VEL
LIN {X 0,Y 267.369,Z 665.007,A -85,B 0,C 180,E1 12774.85,E2 12774.85} C_VEL
LIN {X 0,Y 267.645,Z 658.382,A -85,B 0,C 180,E1 12771.405,E2 12771.405} C_VEL
LIN {X 0,Y 268.3,Z 650.183,A -85,B 0,C 180,E1 12768.172,E2 12768.172} C_VEL
LIN {X 0,Y 269.365,Z 639.869,A -85,B 0,C 180,E1 12764.939,E2 12764.939} C_VEL
LIN {X 0,Y 270.064,Z 634.217,A -85,B 0,C 180,E1 12763.38,E2 12763.38} C_VEL
LIN {X 0,Y 271.734,Z 634.524,A -85,B 0,C 180,E1 12762.438,E2 12762.438} C_VEL
LIN {X 0,Y 274.367,Z 633.985,A -85,B 0,C 180,E1 12761.515,E2 12761.515} C_VEL
LIN {X 0,Y 277.259,Z 633.786,A -85,B 0,C 180,E1 12760.404,E2 12760.404} C_VEL
LIN {X 0,Y 279.438,Z 633.409,A -85,B 0,C 180,E1 12759.691,E2 12759.691} C_VEL
LIN {X 0,Y 283.384,Z 632.704,A -85,B 0,C 180,E1 12758.472,E2 12758.472} C_VEL
LIN {X 0,Y 289.413,Z 631.484,A -85,B 0,C 180,E1 12756.805,E2 12756.805} C_VEL
LIN {X 0,Y 295.931,Z 630.063,A -85,B 0,C 180,E1 12755.23,E2 12755.23} C_VEL
LIN {X 0,Y 303.766,Z 628.045,A -85,B 0,C 180,E1 12753.617,E2 12753.617} C_VEL
LIN {X 0,Y 309.749,Z 626.384,A -85,B 0,C 180,E1 12752.509,E2 12752.509} C_VEL
LIN {X 0,Y 302.691,Z 641.829,A -85,B 0,C 180,E1 12749.861,E2 12749.861} C_VEL
LIN {X 0,Y 295.346,Z 656.658,A -85,B 0,C 180,E1 12746.74,E2 12746.74} C_VEL
LIN {X 0,Y 288.321,Z 670.167,A -85,B 0,C 180,E1 12743.234,E2 12743.234} C_VEL
LIN {X 0,Y 282.211,Z 681.586,A -85,B 0,C 180,E1 12739.581,E2 12739.581} C_VEL
LIN {X 0,Y 276.6,Z 692.084,A -85,B 0,C 180,E1 12735.408,E2 12735.408} C_VEL
LIN {X 0,Y 271.975,Z 701.084,A -85,B 0,C 180,E1 12730.873,E2 12730.873} C_VEL
LIN {X 0,Y 268.507,Z 708.43,A -85,B 0,C 180,E1 12726.041,E2 12726.041} C_VEL
LIN {X 0,Y 266.259,Z 713.908,A -85,B 0,C 180,E1 12721.107,E2 12721.107} C_VEL
LIN {X 0,Y 265.104,Z 717.383,A -85,B 0,C 180,E1 12716.427,E2 12716.427} C_VEL
LIN {X 0,Y 264.612,Z 719.272,A -85,B 0,C 180,E1 12711.968,E2 12711.968} C_VEL
LIN {X 0,Y 264.455,Z 719.839,A -85,B 0,C 180,E1 12707.606,E2 12707.606} C_VEL
LIN {X 0,Y 264.494,Z 719.012,A -85,B 0,C 180,E1 12703.333,E2 12703.333} C_VEL
LIN {X 0,Y 264.761,Z 716.816,A -85,B 0,C 180,E1 12698.908,E2 12698.908} C_VEL
LIN {X 0,Y 265.504,Z 713.287,A -85,B 0,C 180,E1 12694.536,E2 12694.536} C_VEL
LIN {X 0,Y 266.99,Z 707.99,A -85,B 0,C 180,E1 12690,E2 12690} C_VEL
LIN {X 0,Y 269.375,Z 701.024,A -85,B 0,C 180,E1 12685.53,E2 12685.53} C_VEL
LIN {X 0,Y 272.813,Z 692.295,A -85,B 0,C 180,E1 12681.146,E2 12681.146} C_VEL
LIN {X 0,Y 277.338,Z 681.591,A -85,B 0,C 180,E1 12676.872,E2 12676.872} C_VEL
LIN {X 0,Y 282.398,Z 669.963,A -85,B 0,C 180,E1 12673.123,E2 12673.123} C_VEL
LIN {X 0,Y 288,Z 656.985,A -85,B 0,C 180,E1 12669.686,E2 12669.686} C_VEL
LIN {X 0,Y 294.02,Z 642.619,A -85,B 0,C 180,E1 12666.555,E2 12666.555} C_VEL
LIN {X 0,Y 300.457,Z 626.157,A -85,B 0,C 180,E1 12663.624,E2 12663.624} C_VEL
LIN {X 0,Y 306.815,Z 608.444,A -85,B 0,C 180,E1 12661.057,E2 12661.057} C_VEL
LIN {X 0,Y 312.647,Z 590.204,A -85,B 0,C 180,E1 12658.904,E2 12658.904} C_VEL
LIN {X 0,Y 317.331,Z 573.493,A -85,B 0,C 180,E1 12657.283,E2 12657.283} C_VEL
LIN {X 0,Y 318.352,Z 567.77,A -85,B 0,C 180,E1 12656.695,E2 12656.695} C_VEL
LIN {X 0,Y 318.134,Z 554.933,A -85,B 0,C 180,E1 12655.081,E2 12655.081} C_VEL
LIN {X 0,Y 318.285,Z 547.27,A -85,B 0,C 180,E1 12654.267,E2 12654.267} C_VEL
LIN {X 0,Y 318.787,Z 543.221,A -85,B 0,C 180,E1 12653.959,E2 12653.959} C_VEL
LIN {X 0,Y 322.373,Z 522.467,A -85,B 0,C 180,E1 12652.835,E2 12652.835} C_VEL
LIN {X 0,Y 325.041,Z 501.135,A -85,B 0,C 180,E1 12651.97,E2 12651.97} C_VEL
LIN {X 0,Y 331.52,Z 446.719,A -85,B 0,C 180,E1 12650.275,E2 12650.275} C_VEL
LIN {X 0,Y 339.877,Z 372.619,A -85,B 0,C 180,E1 12648.301,E2 12648.301} C_VEL
LIN {X 0,Y 344.384,Z 324.724,A -85,B 0,C 180,E1 12647.147,E2 12647.147} C_VEL
LIN {X 0,Y 334.037,Z 311.573,A -85,B 0,C 180,E1 12643.832,E2 12643.832} C_VEL
LIN {X 0,Y 325.147,Z 301.372,A -85,B 0,C 180,E1 12640.687,E2 12640.687} C_VEL
LIN {X 0,Y 318.35,Z 294.266,A -85,B 0,C 180,E1 12637.995,E2 12637.995} C_VEL
LIN {X 0,Y 314.584,Z 290.462,A -85,B 0,C 180,E1 12636.354,E2 12636.354} C_VEL
LIN {X 0,Y 308.823,Z 284.956,A -85,B 0,C 180,E1 12633.618,E2 12633.618} C_VEL
LIN {X 0,Y 305.526,Z 282.172,A -85,B 0,C 180,E1 12631.796,E2 12631.796} C_VEL
LIN {X 0,Y 304.702,Z 279.846,A -85,B 0,C 180,E1 12629.703,E2 12629.703} C_VEL
LIN {X 0,Y 302.76,Z 275.291,A -85,B 0,C 180,E1 12622.321,E2 12622.321} C_VEL
LIN {X 0,Y 302.588,Z 275.217,A -85,B 0,C 180,E1 12616.313,E2 12616.313} C_VEL
LIN {X 0,Y 302.783,Z 275.878,A -85,B 0,C 180,E1 12614.34,E2 12614.34} C_VEL
LIN {X 0,Y 305.025,Z 280.471,A -85,B 0,C 180,E1 12607.345,E2 12607.345} C_VEL
LIN {X 0,Y 307.275,Z 285.234,A -85,B 0,C 180,E1 12603.172,E2 12603.172} C_VEL
LIN {X 0,Y 309.549,Z 290.222,A -85,B 0,C 180,E1 12599.816,E2 12599.816} C_VEL
LIN {X 0,Y 311.766,Z 295.108,A -85,B 0,C 180,E1 12597.059,E2 12597.059} C_VEL
LIN {X 0,Y 314.695,Z 301.307,A -85,B 0,C 180,E1 12593.973,E2 12593.973} C_VEL
LIN {X 0,Y 319.151,Z 311.803,A -85,B 0,C 180,E1 12589.714,E2 12589.714} C_VEL
LIN {X 0,Y 323.595,Z 323.215,A -85,B 0,C 180,E1 12585.872,E2 12585.872} C_VEL
LIN {X 0,Y 328.157,Z 335.793,A -85,B 0,C 180,E1 12582.261,E2 12582.261} C_VEL
LIN {X 0,Y 329.992,Z 341.432,A -85,B 0,C 180,E1 12580.808,E2 12580.808} C_VEL
LIN {X 0,Y 323.993,Z 368.849,A -85,B 0,C 180,E1 12577.693,E2 12577.693} C_VEL
LIN {X 0,Y 321.159,Z 391.119,A -85,B 0,C 180,E1 12574.865,E2 12574.865} C_VEL
LIN {X 0,Y 325.338,Z 413.011,A -85,B 0,C 180,E1 12572.772,E2 12572.772} C_VEL
LIN {X 0,Y 331.383,Z 435.79,A -85,B 0,C 180,E1 12570.338,E2 12570.338} C_VEL
LIN {X 0,Y 338.091,Z 455.629,A -85,B 0,C 180,E1 12567.988,E2 12567.988} C_VEL
LIN {X 0,Y 339.329,Z 459.379,A -85,B 0,C 180,E1 12567.559,E2 12567.559} C_VEL
LIN {X 0,Y 335.063,Z 482.3,A -85,B 0,C 180,E1 12567.29,E2 12567.29} C_VEL
LIN {X 0,Y 331.14,Z 503.626,A -85,B 0,C 180,E1 12566.75,E2 12566.75} C_VEL
LIN {X 0,Y 325.77,Z 531.983,A -85,B 0,C 180,E1 12565.651,E2 12565.651} C_VEL
LIN {X 0,Y 319.275,Z 559.905,A -85,B 0,C 180,E1 12564.288,E2 12564.288} C_VEL
LIN {X 0,Y 312.921,Z 584.992,A -85,B 0,C 180,E1 12562.713,E2 12562.713} C_VEL
LIN {X 0,Y 306.306,Z 608.983,A -85,B 0,C 180,E1 12560.828,E2 12560.828} C_VEL
LIN {X 0,Y 300.16,Z 629.639,A -85,B 0,C 180,E1 12558.835,E2 12558.835} C_VEL
LIN {X 0,Y 293.948,Z 648.629,A -85,B 0,C 180,E1 12556.57,E2 12556.57} C_VEL
